// TwinCAT 3 PLC project XtsTransport
// Title: XTS Transport
// Author: D.Hauer
// ProjectVersion: 0.0.1
// Description: basic functionblocks for building XTS transport
// ProgramVersion: 3.1.4026.16
// libraries:
//   Tc2_Math, * (Beckhoff Automation GmbH)
//   Tc2_MC2, * (Beckhoff Automation GmbH)
//   Tc2_Standard, * (Beckhoff Automation GmbH)
//   Tc2_System, * (Beckhoff Automation GmbH)
//   Tc2_Utilities, * (Beckhoff Automation GmbH)
//   Tc2_XmlDataSrv, * (Beckhoff Automation GmbH)
//   Tc3_McCollisionAvoidance, * (Beckhoff Automation GmbH)
//   Tc3_McCoordinatedMotion, * (Beckhoff Automation GmbH)
//   Tc3_Module, * (Beckhoff Automation GmbH)
//   Tc3_XTS_Utility, * (Beckhoff Automation GmbH)
//   VisuDialogs, * (System)
// project tree:
//   APPLICATION/ MAIN_APP.TcPOU, fb_Simulation.TcPOU, GVL_APPLICATION.TcGVL
//   APPLICATION/_types/ E_PROCESS_CHECK.TcDUT (not stored), E_PROCESS_CTRL.TcDUT, E_PROCESS_STATE.TcDUT (not stored), ST_PROCESS_CTRL.TcDUT, ST_PROCESS_STATE.TcDUT (not stored), T_PROCESS.TcDUT
//   APPLICATION/_types/fb_Instance/ E_INSTANCE_CHECK.TcDUT (not stored), E_INSTANCE_STATE.TcDUT, fb_Instance.TcPOU
//   APPLICATION/_types/LinkedList/ fb_Process_LinkedListCtrl.TcPOU, I_Process_LinkedList.TcIO (not stored), ST_PROCESS_DATA.TcDUT (not stored), ST_PROCESS_LIST_RESULT.TcDUT
//   / GlobalTextList.TcGTLO (not stored), MAIN.TcPOU, PlcTask.TcTTO
//   MSG/ fb_LocalTime.TcPOU (not stored), f_MessageSet.TcPOU (not stored), GVL_MSG.TcGVL, MessageData.TcPOU, T_MESSAGE_LIST.TcVIS
//   MSG/types/ e_Device.TcDUT, E_MessageType.TcDUT (not stored), E_MESSAGE_STATE.TcDUT (not stored), e_Subdevice.TcDUT, ST_Message.TcDUT (not stored), TL_E_MESSAGETYPE.TcTLO (not stored)
//   XML/Configuration/ fb_Configuration.TcPOU
//   XML/Configuration/types/ E_CONFIG_CTRL.TcDUT (not stored), E_CONFIG_STATE.TcDUT (not stored), fb_XmlRead.TcPOU (not stored), fb_XmlWrite.TcPOU (not stored), ST_Configuration.TcDUT (not stored)
//   XTS/CaGroup/ FB_CaGroup.TcPOU, I_XtsTransport_CaGroup.TcIO (not stored)
//   XTS/CaGroup/types/ E_CA_GROUP_STATE.TcDUT (not stored), E_GROUP_CHECK.TcDUT (not stored), ST_GROUP_INFO.TcDUT (not stored)
//   XTS/ GVL_XTS.TcGVL, XTS_Parameter.TcGVL
//   XTS/Mover/ fb_Mover.TcPOU, fb_MoverCtrl.TcPOU (not stored), I_XtsTransport_Mover.TcIO
//   XTS/Mover/types/ E_MOVER_CTRL.TcDUT (not stored), E_MOVER_STATE.TcDUT (not stored), ST_GEAR_DATA.TcDUT (not stored), ST_MOVER_CTRL.TcDUT (not stored), ST_MOVER_INFO.TcDUT (not stored), ST_MOVER_STATE.TcDUT (not stored), ST_MOVE_DATA.TcDUT (not stored)
//   XTS/XtsStation/ fb_Station.TcPOU, I_XtsTransport_Station.TcIO (not stored)
//   XTS/XtsStation/_types/ E_STATION_CTRL.TcDUT (not stored), E_STATION_STATE.TcDUT (not stored), fb_Station_LinkedListCtrl.TcPOU (not stored), I_Station_LinkedList.TcIO (not stored), ST_STATION_CTRL.TcDUT (not stored), ST_STATION_LIST_RESULT.TcDUT (not stored), ST_STATION_MOVER_DATA.TcDUT (not stored), ST_STATION_PARAMETER.TcDUT (not stored), ST_STATION_STATE.TcDUT (not stored), T_NEST_OFFSET.TcDUT (not stored)
//   XTS/_Visualization/ GROUP_VISU.TcVIS, MOVER_VISU.TcVIS, STATION_VISU.TcVIS, Visualization Manager.TcVMO (not stored), XTS_TRANSPORT.TcVIS, XPU_VISU.TcVIS
//   XTS/_Visualization/textlists/ TL_E_CTRL_MOVER.TcTLO (not stored), TL_E_CTRL_STATION.TcTLO (not stored), TL_E_CTRL_TRANSPORT.TcTLO (not stored), TL_E_CTRL_XPU.TcTLO (not stored)
//   XTS/Xpu/ fb_Xpu.TcPOU (not stored), fb_XpuCtrl.TcPOU (not stored)
//   XTS/Xpu/types/ E_XPU_CHECK.TcDUT (not stored), E_XPU_CTRL.TcDUT (not stored), E_XPU_INIT.TcDUT (not stored), E_XPU_STATE.TcDUT (not stored), ST_XPU_CTRL.TcDUT (not stored), ST_XPU_INFO.TcDUT (not stored), ST_XPU_STATE.TcDUT (not stored)
//   XTS/XtsTransportUnit/ fb_TransportUnit.TcPOU
//   XTS/XtsTransportUnit/types/ E_XTS_TRANSPORT_CHECK.TcDUT (not stored), E_XTS_TRANSPORT_CTRL.TcDUT (not stored), E_XTS_TRANSPORT_STATE.TcDUT, ST_XTS_TRANSPORT_CTRL.TcDUT (not stored), ST_XTS_TRANSPORT_STATE.TcDUT (not stored)
//   XTS/_types/ E_PROGRESS.TcDUT, f_GetProgress.TcPOU (not stored), f_GetState.TcPOU (not stored)

CONFIGURATION XtsTransport
    RESOURCE PLC ON TwinCAT3
        TASK PlcTask(INTERVAL := T#1ms, PRIORITY := 15);
        PROGRAM MAIN WITH PlcTask : MAIN;
        PROGRAM MAIN_APP WITH PlcTask : MAIN_APP;
    END_RESOURCE
END_CONFIGURATION

// ---- APPLICATION/_types/E_PROCESS_CTRL.TcDUT
{attribute 'qualified_only'}
{attribute 'strict'}
{attribute 'to_string'}
TYPE E_PROCESS_CTRL :
(
  PROCESS_INIT              := 10,
  PROCESS_DISABLE           := 20,
  PROCESS_ENABLE            := 30,

  PROCESS_STATIONS_ENTER    := 40,
  PROCESS_STATIONS_SEND,

  PROCESS_START             := 60,
  PROCESS_DONE              := 70,
  PROCESS_STATIONS_OUTFEED  := 80
);
END_TYPE

// ---- APPLICATION/_types/fb_Instance/E_INSTANCE_STATE.TcDUT
{attribute 'qualified_only'}
{attribute 'strict'}
{attribute 'to_string'}
TYPE E_INSTANCE_STATE :
(
	INVALID,
  INIT,
  DISABLED,
  DETECT_IN_LIST,
  ENABLED,
  WORKING,
  FINISH
);
END_TYPE

// ---- APPLICATION/_types/LinkedList/ST_PROCESS_LIST_RESULT.TcDUT
TYPE ST_PROCESS_LIST_RESULT :
STRUCT
  wState    : WORD;   // wState == 0 --> all ok
  nIndex    : ULINT;
  stData    : ST_PROCESS_DATA;  // copy of list entry
END_STRUCT
END_TYPE

// ---- APPLICATION/_types/ST_PROCESS_CTRL.TcDUT
TYPE ST_PROCESS_CTRL :
STRUCT
  Cmd               : E_PROCESS_CTRL;
  ProcessTarget     : UINT;
  ActivateStation   : WORD; // every bit is a XtsStation
  NestMask          : WORD; // every bit is a PosStop in a XtsStation, one mask for all XtsStations
END_STRUCT
END_TYPE

// ---- APPLICATION/_types/T_PROCESS.TcDUT
TYPE T_PROCESS : WORD; END_TYPE

// ---- MSG/types/e_Device.TcDUT
{attribute 'to_string'}
TYPE e_Device :
(
  Device_Null,
  General           :=  1000,
  CaGroup           :=  2000,
  Xpu               :=  3000,
  XpuCtrl           :=  4000,
  Mover             :=  5000,
  MoverCtrl         :=  6000,
  XtsTransportUnit  :=  7000,
  XfcTriggerBox     :=  8000,
  XfcTouchProbe     :=  9000,
  XtsStation        := 10000,

  Camming           := 11000,
  NciChannel        := 12000,
  NciChannelCtrl    := 13000,
  Axis              := 14000,
  XfcAxis           := 15000,
  Data              := 16000,

  Process           := 20000,
  Application       := 30000
)UDINT;
END_TYPE

// ---- MSG/types/e_Subdevice.TcDUT
{attribute 'strict'}
{attribute 'to_string'}
TYPE e_Subdevice :
(
  // sub device for message system
  General                 :=  0,
  // Motion Control FB Instances
  fbPower,
  fbReset,
  fbResetSercos,
  fbHalt,
  fbStop,                 // 5
  fbHome,
  fbJog,
  fbMoveVelocity1,
  fbMoveVelocity2,
  fbMoveAbsolute1,        // 10
  fbMoveAbsolute2,
  fbMoveEndless,
  fbMovePtP,

  // CA CollisionAvoidance FB instances
  // CA group fb instances
  fbCaGroup             := 30,
  fbMoveToPosCa,
  fbSendToAbsPosCa,
  fbSendToModuloPosCa,
  fbGearInPosCa,
  fbGroupAddAxis,
  fbGroupRemoveAxis,
  fbGroupDisable,
  fbGroupEnable,
  fbGroupErrorRead,
  fbGroupStatusRead,
  fbGroupReset,
  fbGroupStop,

  fbGearIn                := 50,
  fbGearOut,
  fbGearInMultiMaster,

  fbCamIn                 := 60,
  fbCamOut,

  fbCamOutV2              := 80,
  fbCamInV2,
  fbCamScalingV2,
  fbCamInfoV2,
  fbReadMotionFunction,
  fbReadMotionFunctionPoint,
  fbReadMotionFunctionValues,
  fbWriteMotionFunction,
  fbWriteMotionFunctionPoint,
  fbSetOnlineChangeMode,

  fbReadParameter         := 100,
  fbReadBoolParameter,
  fbWriteParameter,
  fbWriteBoolParameter,

  fbBuildGroup            := 200,
  fbClearGroup,
  fbLoadProg,
  fbResetItp,
  fbStartStopItp,
  fbEStopItp,             // 205
  fbStepOnAfterEStopItp,
  fbConfirmHskItp,
  fbDelDtgItp,
  fbNciFeedTablePreparation,
  fbNciFeedTable,         // 210
  fbReadLine,
  fbItpReadRParams,
  fbItpWriteRParams,
  Get_ItpState,
  Get_Error,              // 215


  XfcPositionAtTime       := 300,
  XfcTimeOfPosition,
  XfcTimeToPosition,
  XfcTimeToModuloPosition,
  XfcRecordedPosition,
  XfcTouchProbe,          // 305
  XfcTouchProbeEL1258,
  XfcTouchProbeOptions,
  XfcTriggerRef,
  XfcTriggerRef_MT,
  XfcEl1258Interface_MT,  // 310
  XfcRecordedPosition_MT,
  XfcTriggerOut,
  XfcTriggerStart,
  XfcSwitchOn_2252,
  XfcSwitchOff_2252,      // 315
  XfcInit,
  XfcLatchPosition,
  XfcWaitForPosition,

  AxisMode              := 1000,
  AxisControl,

  NciControl            := 2000,
  NciStartUp,
  NciCycle,
  NciIdle,

  StationLinkedList     := 3000,
  StationInitList,
  StationAddHead,
  StationAddTail,
  StationGetHead,
  StationRemoveHeadValue,

  StationControl        := 4000,
  StationState, 

  Xpu_fbEnvironment     := 5000,
  Xpu_fbProcessingUnit,
  Xpu_fbXpuPart,
  Xpu_fbXpuTrack,
  Xpu_fbMc2CaGroup,

  Xpu_fbPartModules     := 5500,

  Xpu_fbMoverXpu        := 6000,

  CamControl            := 8000,
  CamStartUp,
  CamCycle,

  Process_StationCollector    := 11000,
  Process_Process_Collector   := 11100,
  Process_ProcessCollector_Init,
  Process_ProcessCollector_Cycle,
  Process_ProcessCollector_Control,

  Process_LinkedList_GetHead,
  Process_LinkedList_RemoveHead,
  Process_LinkedList_AddTail,

  Process_BufferInfeed
)DINT;
END_TYPE

// ---- XTS/XtsTransportUnit/types/E_XTS_TRANSPORT_STATE.TcDUT
{attribute 'to_string'}
TYPE E_XTS_TRANSPORT_STATE :
(
  TRANSPORT_NULL,
  TRANSPORT_INVALID,
  TRANSPORT_INIT            := 10,  // Xpu, Group, Mover initialization: init TcCOM objects, clear errors, clear group, check Xpu data, check mover detection
  TRANSPORT_IDLE,                   // cyclic check for errors, check Xpu data

  TRANSPORT_MOVER_ENABLE    := 20,  // all mover are enabled, checked for ControlLoopClosed
  TRANSPORT_MOVER_DISABLE,          // all mover are disabled
  TRANSPORT_MOVER_HALT_CA,          // all mover standstill

  TRANSPORT_GROUP_CLEAR     := 30,  // halt all movers, clear errors, remove all movers from group, clear group
  TRANSPORT_GROUP_BUILD,            // add all movers to group
  TRANSPORT_GROUP_ENABLE,           // group with movers is enabled
  TRANSPORT_GROUP_STOP,             // CaGroup Stop, CaGroup Reset, All movers halt

  TRANSPORT_START           := 40,  // move all mover[i] to start position
  TRANSPORT_RESTART                 // move all mover[i] to LastPosition[i]
)UINT;
END_TYPE

// ---- XTS/_types/E_PROGRESS.TcDUT
{attribute 'qualified_only'}
//{attribute 'strict'}
{attribute 'to_string'}
TYPE E_PROGRESS :
(
  // progress is used in project to mirror state of requested command/function
  PROGRESS_INVALID,
  PROGRESS_NOT_EXIST      :=   100,
  PROGRESS_INIT           :=  1000,
  PROGRESS_BUSY           :=  2000,
  PROGRESS_PREPARE        :=  3000,
  PROGRESS_STARTUP        :=  4000,
  PROGRESS_CHECK          :=  5000,
  PROGRESS_OCCUPIED       :=  6000,
  PROGRESS_WORKING        :=  7000,
  PROGRESS_STILL_WORKING  :=  8000,
  PROGRESS_ERROR          :=  9000,
  PROGRESS_DONE           := 10000
)UINT;
END_TYPE

// ---- APPLICATION/GVL_APPLICATION.TcGVL
VAR_GLOBAL CONSTANT
  MAX_PROCESS       : UINT := 11;
END_VAR
{attribute 'qualified_only'}
VAR_GLOBAL
  Simulation        : ARRAY[1..MAX_PROCESS] OF fb_Simulation;
END_VAR

// ---- MSG/GVL_MSG.TcGVL
{attribute 'qualified_only'}
VAR_GLOBAL CONSTANT
  //-----------------------------------------------------------------------------
  // file paths for message system
  //  - compiler define option WIN switches to Windows file paths
  //-----------------------------------------------------------------------------
{IF defined (WIN)}
  {info 'WIN folders'}
  LOG_DIR               : STRING  := 'C:\TwinCAT\#MsgFiles\';
  CONFIG_DIR            : STRING  := 'C:\TwinCAT\XPU_PLC_StationConfig\';
{ELSE}
  {info 'BSD folders'}
  LOG_DIR               : STRING  := '/usr/local/etc/TwinCAT/#MsgFiles/';
  CONFIG_DIR            : STRING  := '/usr/local/etc/TwinCAT/XPU_PLC_StationConfig/';
{END_IF}

  LOG_FILE              : STRING  := 'MSG_XtsTransport_';
  CONFIG_FILE           : STRING  := 'Config_XPU_'; // OTCID of fb_Environment is added to name on writing

  MAX_MESSAGE           : UINT    := 200; // max entry in message list
END_VAR
VAR_GLOBAL
  Messages                        : ARRAY[1..MAX_MESSAGE] OF ST_Message;
  MessageIndex                    : UINT := 1; // message index
  MessageError                    : UINT := 0; // error counter

  fbLocalTime                     : fb_LocalTime;
  dtLocalTime                     : DT;
  sLocalTime                      : STRING;

  MessageLevelXpu                 : E_MessageType;
  MessageLevelStations            : ARRAY[1..MAX_STATION] OF E_MessageType;
  MessageLevelMovers              : ARRAY[1..MAX_MOVER]   OF E_MessageType;

  MessageLevelProcess             : ARRAY[1..MAX_PROCESS] OF E_MessageType;

{IF defined (TEST)}
  {info 'TEST logging enabled'}
  MessageLevel                    : E_MessageType := eMessageVerbose; // a lot of messages
{ELSE}
  MessageLevel                    : E_MessageType := eMessageError;    // not as much messages 
{END_IF}

END_VAR

// ---- XTS/GVL_XTS.TcGVL
{attribute 'qualified_only'}
VAR_GLOBAL
  //---------------------------------------------------------------------------
  // XTS Station
  //  - handshakes mover in station with extern control
  //  - station parameters (positions, gap, dyn. constraints, description...)
  StationStart        : ST_STATION_PARAMETER;   // Xts transport is sending all mover to this position (CMD_TRANSPORT_START)
  StationStartIndex   : UINT := 1;              // index of XtsStation where all movers are entered into linked list.

  // station handshaking with mover and extern process
  // station sends mover to target station/WaitPos
  // station adds mover data to LinkedList.AddTail() of target station
  Station             : ARRAY[1..MAX_STATION] OF fb_Station;
  StationList         : ARRAY[1..MAX_STATION] OF fb_Station_LinkedListCtrl;

  StationQueue        : ARRAY[1..MAX_STATION]    OF 
                        ARRAY[1..MAX_LIST_NODES] OF ST_STATION_MOVER_DATA;

  // interface for access to List methods
  StationListItf      : ARRAY[1..MAX_STATION] OF I_Station_LinkedList;

  // interface for access to station methods
  StationCtrlItf      : ARRAY[1..MAX_STATION] OF I_XtsTransport_Station;

  // ctrl / state datafields for extern control
  StationCtrl         : ARRAY[1..MAX_STATION] OF ST_STATION_CTRL;   // control for extern to write
  StationState        : ARRAY[1..MAX_STATION] OF ST_STATION_STATE;  // state for extern to read

  // station parameter
  StationParameter    : ARRAY[1..MAX_STATION] OF ST_STATION_PARAMETER; // XtsStation (fb_Station) positions and dyn constraints

  // static position offsets in stations
  PositionOffset      : ARRAY[1..MAX_STATION] OF T_NEST_OFFSET; // added to PosStop[] in XtsStation


  //---------------------------------------------------------------------------
  // XTS
  // XTS TransportUnit
  //  - handles request for XPU, Group, Mover, StartUp, ReStart
  XtsTransport        : fb_TransportUnit;         // manages members of XTS transport for extern to access

  XtsTransportCtrl    : ST_XTS_TRANSPORT_CTRL;    // control of XTS transport for extern to write
  XtsTransportState   : ST_XTS_TRANSPORT_STATE;   // state   of XTS transport for extern to read


  //---------------------------------------------------------------------------
  // XPU
  // XTS-Utility checks
  // XTS-Utility interfaces for you to use
  Xpu             : fb_XpuCtrl;

  XpuCtrl         : ST_XPU_CTRL;
  XpuState        : ST_XPU_STATE;
  XpuInfo         : ST_XPU_INFO;
  XpuModules      : ARRAY[1..MAX_MODULE] OF Tc3_XTS_Utility.ST_InfoDataView;


  //---------------------------------------------------------------------------
  // Collision avoidance group CA
  //
  // - add mover to group
  // - build group
  // - clear group
  CaGroup         : FB_CaGroup;                   // cyclic check of CaGroup state and errors; carries methods for handling CaGroup
  CaGroupItf      : I_XtsTransport_CaGroup;       // Interface used by fb_TransportUnit

  // cyclic mapping to MOTION/Objects/CaGroup 
  CaGroupRef      : Tc3_McCoordinatedMotion.AXES_GROUP_REF;

  // Info data from CaGroup FB
  CaGroupInfo     : ST_GROUP_INFO;                // cyclic info about CaGroup for fb_TransportUnit to read
  //---------------------------------------------------------------------------

  //---------------------------------------------------------------------------
  // MC2 encapsulation, CA movement
  Mover           : ARRAY[1..MAX_MOVER] OF fb_MoverCtrl;    // MC and CA methods for mover; cyclic check for individual command on mover

  MoverCtrl       : ARRAY[1..MAX_MOVER] OF ST_MOVER_CTRL;   // control of individual mover for extern to write
  MoverState      : ARRAY[1..MAX_MOVER] OF ST_MOVER_STATE;  // state   of individual mover for extern to read

  MoverItf        : ARRAY[1..MAX_MOVER] OF I_XtsTransport_Mover;  // Interface used by fb_TransportUnit

  LastPosition    : ARRAY[1..MAX_MOVER] OF LREAL;           // on execute of any movement, value is saved here (used by fb_Mover)
  LastGap         : ARRAY[1..MAX_MOVER] OF LREAL;           // on execute of any movement, value is saved here (used by fb_Mover)

  MoverInfo       : ARRAY[1..MAX_MOVER] OF ST_MOVER_INFO;   // cyclic info about mover for extern to read

  MoveData        : ARRAY[1..MAX_MOVER] OF ST_MOVE_DATA;    // dynamic constraints for move commands
  GearData        : ARRAY[1..MAX_MOVER] OF ST_GEAR_DATA;    // dynamic constraints and positions for GearIn/GearInPosCa
  
  // cyclic mapping to MOTION/Axes
  AxisRefMover    : ARRAY[1..MAX_MOVER] OF Tc2_MC2.AXIS_REF;
  //---------------------------------------------------------------------------

  //---------------------------------------------------------------------------
  // XML configuration helper
  XmlConfiguration   : fb_Configuration;


END_VAR

// ---- XTS/XTS_Parameter.TcGVL
//{attribute 'qualified_only'}
VAR_GLOBAL CONSTANT
// HAUD 2025 08 09
//
//    XTS_TRANSPORT_LAYER project
//    
//    MIT License
//    
//    Copyright (c) 2025 HAUD
//    
//    Permission is hereby granted, free of charge, to any person obtaining a copy
//    of this software and associated documentation files (the "Software"), to deal
//    in the Software without restriction, including without limitation the rights
//    to use, copy, modify, merge, publish, distribute, sublicense, and/or sell
//    copies of the Software, and to permit persons to whom the Software is
//    furnished to do so, subject to the following conditions:
//    
//    The above copyright notice and this permission notice shall be included in all
//    copies or substantial portions of the Software.
//    
//    THE SOFTWARE IS PROVIDED "AS IS", WITHOUT WARRANTY OF ANY KIND, EXPRESS OR
//    IMPLIED, INCLUDING BUT NOT LIMITED TO THE WARRANTIES OF MERCHANTABILITY,
//    FITNESS FOR A PARTICULAR PURPOSE AND NONINFRINGEMENT. IN NO EVENT SHALL THE
//    AUTHORS OR COPYRIGHT HOLDERS BE LIABLE FOR ANY CLAIM, DAMAGES OR OTHER
//    LIABILITY, WHETHER IN AN ACTION OF CONTRACT, TORT OR OTHERWISE, ARISING FROM,
//    OUT OF OR IN CONNECTION WITH THE SOFTWARE OR THE USE OR OTHER DEALINGS IN THE
//    SOFTWARE.

  Version             : STRING  := '4.00.11';

  MAX_MOVER           : UINT    := TO_UINT(Tc3_XTS_Utility.TcIoXtsEnvironmentParameterList.MaxXtsMoversPerXpu);
  MAX_MODULE          : UINT    := TO_UINT(Tc3_XTS_Utility.TcIoXtsEnvironmentParameterList.MaxModulesPerPart);
  MAX_PART            : UINT    := TO_UINT(Tc3_XTS_Utility.TcIoXtsEnvironmentParameterList.MaxXtsPartsPerXpu);
  MAX_TRACK           : UINT    := TO_UINT(Tc3_XTS_Utility.TcIoXtsEnvironmentParameterList.MaxXtsTracksPerXpu);
  MAX_GROUP           : UINT    := TO_UINT(Tc3_XTS_Utility.TcIoXtsEnvironmentParameterList.MaxXtsCaGroup);

  MAX_INFO_SERVER     : UINT    := TO_UINT(Tc3_XTS_Utility.TcIoXtsEnvironmentParameterList.MaxXtsInfoServer);
  MAX_INFO_STATION    : UINT    := TO_UINT(Tc3_XTS_Utility.TcIoXtsEnvironmentParameterList.MaxXtsInfoStation);
  MAX_INFO_STOP_POS   : UINT    := TO_UINT(Tc3_XTS_Utility.TcIoXtsEnvironmentParameterList.MaxXtsStopPositionsPerStation);

  MAX_PARAMETER_SET   : UINT    := TO_UINT(Tc3_XTS_Utility.TcIoXtsEnvironmentParameterList.MaxXtsParameterSet);

  MAX_NCT_BASE_UNIT   : UINT    := TO_UINT(Tc3_XTS_Utility.TcIoXtsEnvironmentParameterList.MaxXtsNctBaseUnitInterfaces);

  MAX_STATION         : UINT    := 22;

  MAX_STATION_NEST    : UINT    := TO_UINT(SIZEOF(ST_STATION_STATE.nMask)*8);
  // MAX_LIST_NODES      : UINT    := MAX_MOVER;
  MAX_LIST_NODES      : UINT    := 32; // visualization can not handle access to MAX_MOVER
  MAX_MASTER          : UINT    := 1;
END_VAR

// ---- XTS/Mover/I_XtsTransport_Mover.TcIO
INTERFACE I_XtsTransport_Mover

METHOD Disable : E_PROGRESS
VAR_INPUT
  Execute             : BOOL;
END_VAR
END_METHOD

METHOD Enable : E_PROGRESS
VAR_INPUT
  Execute             : BOOL;
END_VAR
END_METHOD

METHOD GearIn : E_PROGRESS;
VAR_INPUT
  Execute             : BOOL;
  stMoveData          : ST_MOVE_DATA;
  stGearData          : ST_GEAR_DATA;
END_VAR
END_METHOD

METHOD GearInPosCa : E_PROGRESS
VAR_INPUT
  Execute             : BOOL;
  stMoveData          : ST_MOVE_DATA;
  stGearData          : ST_GEAR_DATA;  
END_VAR
END_METHOD

METHOD GearOut : E_PROGRESS
VAR_INPUT
  Execute             : BOOL;
END_VAR
END_METHOD

METHOD Halt : E_PROGRESS
VAR_INPUT
  Execute             : BOOL;
  stMoveData          : ST_MOVE_DATA;
END_VAR
END_METHOD

METHOD HaltCa : E_PROGRESS
VAR_INPUT
  Execute             : BOOL;
  stMoveData          : ST_MOVE_DATA;
END_VAR
END_METHOD

PROPERTY MessageLevel : e_messagetype
SET
END_SET
END_PROPERTY

PROPERTY ModuloTurn : dint
GET
END_GET
END_PROPERTY

METHOD MoveToPos : E_PROGRESS
VAR_INPUT
  Execute             : BOOL;
  stMoveData          : ST_MOVE_DATA;
END_VAR
END_METHOD

METHOD MoveToPosCa : E_PROGRESS
VAR_INPUT
  Execute             : BOOL;
  stMoveData          : ST_MOVE_DATA;
END_VAR
END_METHOD

PROPERTY RailLength : LREAL
GET
END_GET
SET
END_SET
END_PROPERTY

METHOD Reset : E_PROGRESS
VAR_INPUT
  Execute             : BOOL;
END_VAR
END_METHOD

METHOD SendToAbsPosCa : E_PROGRESS
VAR_INPUT
  Execute             : BOOL;
  stMoveData          : ST_MOVE_DATA;
END_VAR
END_METHOD

METHOD SendToModuloPosCa : E_PROGRESS
VAR_INPUT
  Execute             : BOOL;
  stMoveData          : ST_MOVE_DATA;
END_VAR
END_METHOD

METHOD Stop : E_PROGRESS
VAR_INPUT
  Execute             : BOOL;
  stMoveData          : ST_MOVE_DATA;
END_VAR
END_METHOD

END_INTERFACE

// ---- MAIN.TcPOU
//---------------------------------------------------------------------------------------------------------------
//
//  HAUD 2024.03.18
//
//  - XTS_TRANSPORT_LAYER
//  - transport layer members:
//    - CaGroup
//      - access to Group functions
//
//    - Mover
//      - access to MC and CA motion functions
//
//    - Xpu (ProcessingUnit)
//      - access to TcCOM Objects in Environment
//
//    - Transport Control Unit
//      - coordinates members to get XTS in defined states
//
//    - Xts Stations
//      - handshakes with extern control for mover transport
//
//  - global datafields for mrmbers in GVL_XTS namespace
//  - global interface datafields for use in members
//  - structures are assigned by reference for every member
//
//---------------------------------------------------------------------------------------------------------------
// HAUD 2024 05 29
//
//    XTS_TRANSPORT_LAYER project
//    
//    MIT License
//    
//    Copyright (c) 2024 HAUD
//    
//    Permission is hereby granted, free of charge, to any person obtaining a copy
//    of this software and associated documentation files (the "Software"), to deal
//    in the Software without restriction, including without limitation the rights
//    to use, copy, modify, merge, publish, distribute, sublicense, and/or sell
//    copies of the Software, and to permit persons to whom the Software is
//    furnished to do so, subject to the following conditions:
//    
//    The above copyright notice and this permission notice shall be included in all
//    copies or substantial portions of the Software.
//    
//    THE SOFTWARE IS PROVIDED "AS IS", WITHOUT WARRANTY OF ANY KIND, EXPRESS OR
//    IMPLIED, INCLUDING BUT NOT LIMITED TO THE WARRANTIES OF MERCHANTABILITY,
//    FITNESS FOR A PARTICULAR PURPOSE AND NONINFRINGEMENT. IN NO EVENT SHALL THE
//    AUTHORS OR COPYRIGHT HOLDERS BE LIABLE FOR ANY CLAIM, DAMAGES OR OTHER
//    LIABILITY, WHETHER IN AN ACTION OF CONTRACT, TORT OR OTHERWISE, ARISING FROM,
//    OUT OF OR IN CONNECTION WITH THE SOFTWARE OR THE USE OR OTHER DEALINGS IN THE
//    SOFTWARE.
//---------------------------------------------------------------------------------------------------------------
PROGRAM MAIN
VAR
	bInit 				: BOOL;
  eInit         : E_PROGRESS;

  nStation,
	nMover,
  nMoverSelected,
  nStationSelected,
  nStationParameter   : UINT;

  sStationText        : STRING(30);

  eTransportState     : E_XTS_TRANSPORT_STATE;
  eTransportResult    : E_PROGRESS;

  eXpuState           : E_XPU_STATE;
  eXpuResult          : E_PROGRESS;
  eXpuCheck           : E_XPU_CHECK;

  eMoverState         : E_MOVER_STATE;
  eMoverResult        : E_PROGRESS;

  sCaGroupState,
  sTransportState,
  sTransportCheck,
  sTransportResult,
  sXpuState,
  sXpuResult,
  sXpuCheck,
  sXpuOpMode,
  sXpuMoverdetectionMode,
  sXpuMoverAssignement,
  sMoverState,
  sMoverResult,
  sStationState,
  sStationStateMask,
  sStationCtrlMask        : STRING;

  bStationEnable,
  bStationEnter,
  bStationStart,
  bStationDone,
  bStationOut,
  bStationGone            : BOOL;

  tStationSelectedQueue   : ARRAY[1..MAX_LIST_NODES] OF ST_STATION_MOVER_DATA;

  tonWriteLog             : Tc2_Standard.TON;
  tWriteLog               : TIME := T#5S;

  nStn                    : UINT;
END_VAR

//############################################################################
// Local time; used for timestamps
//############################################################################
GVL_MSG.fbLocalTime(
                    sLocalTime          => GVL_MSG.sLocalTime, 
                    dtLocalTime         => GVL_MSG.dtLocalTime);
//############################################################################

//############################################################################
// 	example for init sequence
//############################################################################	
IF NOT bInit
THEN
  CASE eInit
  OF
    E_PROGRESS.PROGRESS_INVALID,
    E_PROGRESS.PROGRESS_DONE:         // clear command interface
      eInit                                   := E_PROGRESS.PROGRESS_BUSY;
      GVL_XTS.XpuCtrl.Cmd                     := E_XPU_CTRL.XTS_CMD_NULL;
      GVL_MSG.MessageLevelXpu                 := GVL_MSG.MessageLevel;
      GVL_XTS.CaGroup.MessageLevel            := GVL_MSG.MessageLevel;
      FOR nStation := 1 TO MAX_STATION
      DO
        GVL_MSG.MessageLevelStations[nStation]:= GVL_MSG.MessageLevel;
      END_FOR
      FOR nMover := 1 TO MAX_MOVER
      DO
        GVL_MSG.MessageLevelMovers[nMover]    := GVL_MSG.MessageLevel;
      END_FOR


    E_PROGRESS.PROGRESS_BUSY:         // init Xpu, ProcessingUnit, MotorModules
      eInit                                   := E_PROGRESS.PROGRESS_PREPARE;
      GVL_XTS.XpuCtrl.Cmd                     := E_XPU_CTRL.XTS_CMD_INIT;

    E_PROGRESS.PROGRESS_PREPARE:      // wait for init to be done
      IF (GVL_XTS.XpuState.State      = E_XPU_STATE.XTS_INIT + E_PROGRESS.PROGRESS_DONE)
      THEN
        eInit                                 := E_PROGRESS.PROGRESS_STARTUP;
        GVL_XTS.XpuCtrl.Cmd                   := E_XPU_CTRL.XTS_IDLE;
      END_IF

    E_PROGRESS.PROGRESS_STARTUP:      // assign mover interfaces
      eInit                                   := E_PROGRESS.PROGRESS_CHECK;
      FOR nMover := 1 TO MAX_MOVER
      DO
        GVL_XTS.MoverItf[nMover]              := GVL_XTS.Mover[nMover];
      END_FOR

    E_PROGRESS.PROGRESS_CHECK:        // assign CaGroup interface
      eInit                                   := E_PROGRESS.PROGRESS_OCCUPIED;
      GVL_XTS.CaGroupItf                      := GVL_XTS.CaGroup;

    E_PROGRESS.PROGRESS_OCCUPIED:     // StartStation for XtsTransportCtrl.Cmd := E_XTS_TRANSPORT_CTRL.CMD_TRANSPORT_START;
      eInit                                   := E_PROGRESS.PROGRESS_WORKING;
      // where to start?
      GVL_XTS.XtsTransport.StationStartIndex  := 1;

      StationParameterInit();


    E_PROGRESS.PROGRESS_WORKING:
      // Start Position parameters
      GVL_XTS.StationStart.rPosWait           :=    GVL_XTS.StationParameter[GVL_XTS.XtsTransport.StationStartIndex].rPosWait -10.0; // this value may differ from the GVL_XTS.StationParameter[StartStationIndex], IF it differs, you MUST have room for positive movement to GVL_XTS.StationParameter[StartStationIndex].rWaitPos
      GVL_XTS.StationStart.rGap               :=    105.0; // may differ, or just copy from GVL_XTS.StationParameter[StartStationIndex]
      GVL_XTS.StationStart.rVelo              :=    750.0; // may differ, or just copy from GVL_XTS.StationParameter[StartStationIndex]
      GVL_XTS.StationStart.rAccDec            :=  12000.0; // may differ, or just copy from GVL_XTS.StationParameter[StartStationIndex]
      GVL_XTS.StationStart.rJerk              := 400000.0; // may differ, or just copy from GVL_XTS.StationParameter[StartStationIndex], the movements are more robust if you keep this value in a narrow range, since jumps lead to adjusting movements within the CA Group

      IF (GVL_XTS.XtsTransport.StationStartIndex > 0) AND
         (GVL_XTS.XtsTransport.StationStartIndex < MAX_STATION+1)
      THEN
        GVL_XTS.StationStart.nConfiguredStopCount := GVL_XTS.StationParameter[GVL_XTS.XtsTransport.StationStartIndex].nConfiguredStopCount;
      END_IF

      bInit                                           := TRUE;
      eInit                                           := E_PROGRESS.PROGRESS_DONE;
  END_CASE
END_IF

//############################################################################
// 	XTS Transport Unit
//############################################################################
//  - main control function block for transport layer
//  - requires access to member controls
//    - Xpu
//    - CaGroup
//    - Mover
//    - Station Control
//    - Station LinkedList Interface
//############################################################################
//
// cyclic call
GVL_XTS.XtsTransport();

// main control
GVL_XTS.XtsTransport.Ctrl               REF= GVL_XTS.XtsTransportCtrl;   // main control
GVL_XTS.XtsTransport.State              REF= GVL_XTS.XtsTransportState;  // main state
                                        
// member controls                      
GVL_XTS.XtsTransport.XpuCtrl            REF= GVL_XTS.XpuCtrl;
GVL_XTS.XtsTransport.XpuState           REF= GVL_XTS.XpuState;
GVL_XTS.XtsTransport.XpuInfo            REF= GVL_XTS.XpuInfo;
                                        
GVL_XTS.XtsTransport.GroupItf           :=   GVL_XTS.CaGroupItf;
GVL_XTS.XtsTransport.GroupInfo          REF= GVL_XTS.CaGroupInfo;
                                        
GVL_XTS.XtsTransport.MoverItf           REF= GVL_XTS.MoverItf;
GVL_XTS.XtsTransport.MoverInfo          REF= GVL_XTS.MoverInfo;
GVL_XTS.XtsTransport.MoverLastPosition  REF= GVL_XTS.LastPosition;
GVL_XTS.XtsTransport.MoverLastGap       REF= GVL_XTS.LastGap;
                                        
GVL_XTS.XtsTransport.StationStart       REF= GVL_XTS.StationStart;      // start position for E_XTS_TRANSPORT_CTRL.CMD_TRANSPORT_START
GVL_XTS.XtsTransport.StationCtrlItf     REF= GVL_XTS.StationCtrlItf;    // station interfaces are required for accessing station methods
GVL_XTS.XtsTransport.StationListsItf    REF= GVL_XTS.StationListItf;    // list interface is required for access to linked list methods
GVL_XTS.XtsTransport.StationControl     REF= GVL_XTS.StationCtrl;
GVL_XTS.XtsTransport.StationState       REF= GVL_XTS.StationState;
//############################################################################



//############################################################################
// 	XTS Stations
//############################################################################	
FOR nStation := 1 TO MAX_STATION
DO
  GVL_XTS.Station[nStation].StationId   := nStation;
  GVL_XTS.Station[nStation].MessageLevel:= GVL_MSG.MessageLevelStations[nStation];

  GVL_XTS.StationListItf[nStation]      := GVL_XTS.StationList[nStation];   // interfaces for list methods
  GVL_XTS.StationCtrlItf[nStation]      := GVL_XTS.Station[nStation];       // interfaces for station methods

  GVL_XTS.Station[nStation].Ctrl        REF= GVL_XTS.StationCtrl;           // station ctrl from extern
  GVL_XTS.Station[nStation].State       REF= GVL_XTS.StationState;          // station state to extern

  GVL_XTS.Station[nStation].ItfStations REF= GVL_XTS.StationListItf;        // give every station all list interfaces for writing mover tickets
  GVL_XTS.Station[nStation].ItfMover    REF= GVL_XTS.MoverItf;              // give every station all mover interfaces for movement in / out of station
  GVL_XTS.Station[nStation].Mover       REF= GVL_XTS.AxisRefMover;          // AXIS_REF to read infos from
  GVL_XTS.Station[nStation].MoverOffset REF= GVL_XTS.PositionOffset;        // static offsets for all stations, all movers, all stop positions


  GVL_XTS.Station[nStation].StationParameter  REF= GVL_XTS.StationParameter;// give every station all station parameters for sending to WaitPos of target station

  // cyclic call
  GVL_XTS.Station[nStation].Cycle();                                        // cycle for handshaking with extern

  // Queue data for each station
  GVL_XTS.StationQueue[nStation]        := GVL_XTS.StationListItf[nStation].Data;
END_FOR
//############################################################################



//############################################################################
// 	XPU environment
//############################################################################	
GVL_XTS.Xpu.XpuInstance               :=   1;
GVL_XTS.Xpu.MessageLevel              :=   GVL_MSG.MessageLevelXpu;

GVL_XTS.Xpu.Ctrl                      REF= GVL_XTS.XpuCtrl;
GVL_XTS.Xpu.State                     REF= GVL_XTS.XpuState;
GVL_XTS.Xpu.XpuModuleInfoData         REF= GVL_XTS.XpuModules;

GVL_XTS.Xpu.CaGroupOID                :=   GVL_XTS.CaGroup.GroupInfo.CaGroupOID;

// cyclic call
GVL_XTS.Xpu();
GVL_XTS.XpuInfo                       :=   GVL_XTS.Xpu.XpuInfo;
//############################################################################


//############################################################################	
// 	CA-Group Class
//############################################################################	
// assignment
GVL_XTS.CaGroup.AxisRef               REF= GVL_XTS.AxisRefMover;
// Interface to Mover methods
GVL_XTS.CaGroup.MoverItf              REF= GVL_XTS.MoverItf; 

GVL_XTS.CaGroup.GroupRef              REF= GVL_XTS.CaGroupRef;

// cyclic call
GVL_XTS.CaGroup.InfoCycle(TRUE); // read group status

// InfoData from group
GVL_XTS.CaGroupInfo                   :=   GVL_XTS.CaGroup.GroupInfo;

// Interface of CaGroup
GVL_XTS.CaGroupItf                    :=   GVL_XTS.CaGroup;
//############################################################################


//############################################################################
// Mover Class	
//############################################################################	
FOR nMover := 1 TO MAX_MOVER
DO
  GVL_XTS.Mover[nMover].MoverId       :=   nMover;
  GVL_XTS.Mover[nMover].RailLength    :=   GVL_XTS.Xpu.RailLength;  // mover needs RailLength, in order to calc absolute position from modulo input
  GVL_XTS.Mover[nMover].MessageLevel  :=   GVL_MSG.MessageLevelMovers[nMover];

  GVL_XTS.Mover[nMover].Ctrl          REF= GVL_XTS.MoverCtrl;       // mover control from extern
  GVL_XTS.Mover[nMover].State         REF= GVL_XTS.MoverState;      // mover state to extern

  GVL_XTS.Mover[nMover].MoveData      REF= GVL_XTS.MoveData;        // dyn constraints for extern to write
  GVL_XTS.Mover[nMover].GearData      REF= GVL_XTS.GearData;        // GearIn/GearInPosCa data fro extern to write

  // assignment	
  GVL_XTS.Mover[nMover].Mover         REF= GVL_XTS.AxisRefMover[nMover];  // axis reference to Mover function block
  GVL_XTS.Mover[nMover].LastGap       REF= GVL_XTS.LastGap[nMover];       // reference to last used gap value datafield
  GVL_XTS.Mover[nMover].LastPosition  REF= GVL_XTS.LastPosition[nMover];  // reference to last position datafield

  GVL_XTS.Mover[nMover].MoverInfo		  REF= GVL_XTS.MoverInfo[nMover];     // refernence to mover info data (ActPos, SetPos, ...)

  GVL_XTS.MoverItf[nMover]            :=   GVL_XTS.Mover[nMover];

  // cyclic call
  GVL_XTS.Mover[nMover].Cycle();  // call AXIS_REF()
  GVL_XTS.Mover[nMover]();        // call Ctrl/State
END_FOR


//############################################################################


//############################################################################
// /logging
//############################################################################
tonWriteLog(IN:= TRUE, PT := tWriteLog);

IF (tonWriteLog.Q)
THEN
  MessageData.bWriteFile      := TRUE;
  tonWriteLog(IN:= FALSE);
END_IF

//-----------------------------------------------------------------------------------------------------------------
// write message list to file
//-----------------------------------------------------------------------------------------------------------------
MessageData(pList			        := ADR(GVL_MSG.Messages),
			      pLocalTime        := ADR(GVL_MSG.dtLocalTime), 
			      bBusy=> );

// clear write trigger
IF MessageData.bWriteFile AND
   MessageData.bDone
THEN
  MessageData.bWriteFile      := FALSE;
END_IF
//############################################################################
// logging/
//############################################################################



//############################################################################
// \xml config 
//    no startup read 
//    for manual use only
//############################################################################
GVL_XTS.XmlConfiguration.StationData   := ADR(GVL_XTS.StationParameter);
GVL_XTS.XmlConfiguration.Identity      := GVL_XTS.Xpu.XpuOtcid;
GVL_XTS.XmlConfiguration();
//############################################################################
// xml config/
//############################################################################


//############################################################################
// Visualization data	
//############################################################################	
// get enumerations from XPU for visu:
eTransportState                       := f_GetState   (GVL_XTS.XtsTransportState.State);
eTransportResult                      := f_GetProgress(GVL_XTS.XtsTransportState.State);

eXpuState                             := f_GetState   (GVL_XTS.XpuState.State);
eXpuResult                            := f_GetProgress(GVL_XTS.XpuState.State);

eXpuCheck                             := GVL_XTS.XpuState.Check;

// display xpu state and result in visu
// get strings and info
sCaGroupState                         := TO_STRING(GVL_XTS.CaGroupInfo.CaGroupState);

sTransportState                       := TO_STRING(eTransportState);
sTransportCheck                       := TO_STRING(GVL_XTS.XtsTransportState.Check);
sTransportResult                      := TO_STRING(eTransportResult);

sXpuState                             := TO_STRING(eXpuState);
sXpuResult                            := TO_STRING(eXpuResult);
sXpuCheck                             := TO_STRING(eXpuCheck);

sXpuOpMode                            := GVL_XTS.Xpu.OpModeToString();
sXpuMoverdetectionMode                := GVL_XTS.Xpu.IdDetectionModeToString();
sXpuMoverAssignement                  := GVL_XTS.Xpu.MoverPositionAssignementToString();

nMoverSelected                        := SEL((nMoverSelected<1), nMoverSelected, 1);
nMoverSelected                        := SEL((nMoverSelected>MAX_MOVER), nMoverSelected, MAX_MOVER);

nStationSelected                      := SEL((nStationSelected<1), nStationSelected, 1);
nStationSelected                      := SEL((nStationSelected>MAX_STATION), nStationSelected, MAX_STATION);

bStationEnable                        := SEL((GVL_XTS.StationCtrl[nStationSelected].eCmd = E_STATION_CTRL.STATION_ENABLE),        FALSE, TRUE);
bStationEnter                         := SEL((GVL_XTS.StationCtrl[nStationSelected].eCmd = E_STATION_CTRL.STATION_MOVER_ENTER),   FALSE, TRUE);
bStationStart                         := SEL((GVL_XTS.StationCtrl[nStationSelected].eCmd = E_STATION_CTRL.STATION_PROCESS_START), FALSE, TRUE);
bStationDone                          := SEL((GVL_XTS.StationCtrl[nStationSelected].eCmd = E_STATION_CTRL.STATION_PROCESS_DONE),  FALSE, TRUE);
bStationOut                           := SEL((GVL_XTS.StationCtrl[nStationSelected].eCmd = E_STATION_CTRL.STATION_MOVER_OUT),     FALSE, TRUE);
bStationGone                          := SEL((GVL_XTS.StationCtrl[nStationSelected].eCmd = E_STATION_CTRL.STATION_MOVER_GONE),    FALSE, TRUE);

eMoverState                           := f_GetState   (GVL_XTS.MoverState[nMoverSelected].State);
eMoverResult                          := f_GetProgress(GVL_XTS.MoverState[nMoverSelected].State);

sMoverState                           := TO_STRING(eMoverState);
sMoverResult                          := TO_STRING(eMoverResult);

sStationState                         := TO_STRING(GVL_XTS.StationState[nStationSelected].eState);
sStationStateMask                     := Tc2_Utilities.BYTE_TO_BINSTR(GVL_XTS.StationState[nStationSelected].nMask, 8);
sStationCtrlMask                      := Tc2_Utilities.BYTE_TO_BINSTR(GVL_XTS.StationCtrl[nStationSelected].nMask, 8);

tStationSelectedQueue                 := GVL_XTS.StationQueue[nStationSelected];

ACTION StationParameterInit:
//---------------------------------------------------------------------------------------
//---------------------------------------------------------------------------------------
//
//
//---------------------------------------------------------------------------------------
//---------------------------------------------------------------------------------------
nStn                    := 1;
GVL_XTS.StationParameter[nStn].sText               := 'STN_12';
GVL_XTS.StationParameter[nStn].rPosWait            :=   6250.0; // absolute modulo position
GVL_XTS.StationParameter[nStn].rPosStop[1]         :=     62.5; // relative to rPosWait
GVL_XTS.StationParameter[nStn].rReleaseDistance    :=     -5.0; // relative to Mover.ActPos

GVL_XTS.StationParameter[nStn].rGap                :=    105.0;
GVL_XTS.StationParameter[nStn].rVelo               :=   1750.0;
GVL_XTS.StationParameter[nStn].rAccDec             :=  17500.0;
GVL_XTS.StationParameter[nStn].rJerk               := 800000.0;
//---------------------------------------------------------------------------------------
//---------------------------------------------------------------------------------------
//
//
//---------------------------------------------------------------------------------------
//---------------------------------------------------------------------------------------
nStn                    := 2;
GVL_XTS.StationParameter[nStn].sText               := 'STN_01(1)';
GVL_XTS.StationParameter[nStn].rPosWait            :=    125.0; // absolute modulo position
GVL_XTS.StationParameter[nStn].rPosStop[1]         :=     62.5; // relative to rPosWait
GVL_XTS.StationParameter[nStn].rReleaseDistance    :=     40.0; // relative to Mover.ActPos

GVL_XTS.StationParameter[nStn].rGap                :=    105.0;
GVL_XTS.StationParameter[nStn].rVelo               :=   2500.0;
GVL_XTS.StationParameter[nStn].rAccDec             :=  17500.0;
GVL_XTS.StationParameter[nStn].rJerk               := 800000.0;

nStn                    := 3;
GVL_XTS.StationParameter[nStn].sText               := 'STN_01(2)';
GVL_XTS.StationParameter[nStn].rPosWait            :=    125.0; // absolute modulo position
GVL_XTS.StationParameter[nStn].rPosStop[1]         :=    187.5; // relative to rPosWait
GVL_XTS.StationParameter[nStn].rReleaseDistance    :=     30.0; // relative to Mover.ActPos

GVL_XTS.StationParameter[nStn].rGap                :=    105.0;
GVL_XTS.StationParameter[nStn].rVelo               :=   2500.0;
GVL_XTS.StationParameter[nStn].rAccDec             :=  17500.0;
GVL_XTS.StationParameter[nStn].rJerk               := 800000.0;

nStn                    := 4;
GVL_XTS.StationParameter[nStn].sText               := 'STN_01(3)';
GVL_XTS.StationParameter[nStn].rPosWait            :=    125.0; // absolute modulo position
GVL_XTS.StationParameter[nStn].rPosStop[1]         :=    312.5; // relative to rPosWait
GVL_XTS.StationParameter[nStn].rReleaseDistance    :=     20.0; // relative to Mover.ActPos

GVL_XTS.StationParameter[nStn].rGap                :=    105.0;
GVL_XTS.StationParameter[nStn].rVelo               :=   2500.0;
GVL_XTS.StationParameter[nStn].rAccDec             :=  17500.0;
GVL_XTS.StationParameter[nStn].rJerk               := 800000.0;

nStn                    := 5;
GVL_XTS.StationParameter[nStn].sText               := 'STN_01(4)';
GVL_XTS.StationParameter[nStn].rPosWait            :=    125.0; // absolute modulo position
GVL_XTS.StationParameter[nStn].rPosStop[1]         :=    437.5; // relative to rPosWait
GVL_XTS.StationParameter[nStn].rReleaseDistance    :=     10.0; // relative to Mover.ActPos

GVL_XTS.StationParameter[nStn].rGap                :=    105.0;
GVL_XTS.StationParameter[nStn].rVelo               :=   2500.0;
GVL_XTS.StationParameter[nStn].rAccDec             :=  17500.0;
GVL_XTS.StationParameter[nStn].rJerk               := 800000.0;
//---------------------------------------------------------------------------------------
//---------------------------------------------------------------------------------------
//
//
//---------------------------------------------------------------------------------------
//---------------------------------------------------------------------------------------
nStn                    := 6;
GVL_XTS.StationParameter[nStn].sText               := 'STN_02(1)';
GVL_XTS.StationParameter[nStn].rPosWait            :=   1140.0; // absolute modulo position

GVL_XTS.StationParameter[nStn].nConfiguredStopCount:=      2;
GVL_XTS.StationParameter[nStn].rPosStop[1]         :=    162.5; // relative to rPosWait
GVL_XTS.StationParameter[nStn].rPosStop[2]         :=    202.5; // relative to rPosWait

GVL_XTS.StationParameter[nStn].rReleaseDistance    :=    150.0; // relative to Mover.ActPos

GVL_XTS.StationParameter[nStn].rGap                :=    105.0;
GVL_XTS.StationParameter[nStn].rVelo               :=   2500.0;
GVL_XTS.StationParameter[nStn].rAccDec             :=  17500.0;
GVL_XTS.StationParameter[nStn].rJerk               := 800000.0;


nStn                    := 7;
GVL_XTS.StationParameter[nStn].sText               := 'STN_02(2)';
GVL_XTS.StationParameter[nStn].rPosWait            :=   1140.0; // absolute modulo position

GVL_XTS.StationParameter[nStn].nConfiguredStopCount:=      2;
GVL_XTS.StationParameter[nStn].rPosStop[1]         :=    268.5; // relative to rPosWait
GVL_XTS.StationParameter[nStn].rPosStop[2]         :=    307.5; // relative to rPosWait

GVL_XTS.StationParameter[nStn].rReleaseDistance    :=    100.0; // relative to Mover.ActPos

GVL_XTS.StationParameter[nStn].rGap                :=    105.0;
GVL_XTS.StationParameter[nStn].rVelo               :=   2500.0;
GVL_XTS.StationParameter[nStn].rAccDec             :=  17500.0;
GVL_XTS.StationParameter[nStn].rJerk               := 800000.0;
//---------------------------------------------------------------------------------------
//---------------------------------------------------------------------------------------
//---------------------------------------------------------------------------------------
//---------------------------------------------------------------------------------------
//
//
//---------------------------------------------------------------------------------------
//---------------------------------------------------------------------------------------
nStn                    := 8;
GVL_XTS.StationParameter[nStn].sText               := 'STN_03';
GVL_XTS.StationParameter[nStn].rPosWait            :=   1675.0; // absolute modulo position
GVL_XTS.StationParameter[nStn].rPosStop[1]         :=     60.5; // relative to rPosWait
GVL_XTS.StationParameter[nStn].rReleaseDistance    :=      2.0; // relative to Mover.ActPos

GVL_XTS.StationParameter[nStn].rGap                :=    105.0;
GVL_XTS.StationParameter[nStn].rVelo               :=    500.0;
GVL_XTS.StationParameter[nStn].rAccDec             :=  17500.0;
GVL_XTS.StationParameter[nStn].rJerk               := 800000.0;
//---------------------------------------------------------------------------------------
//---------------------------------------------------------------------------------------
//---------------------------------------------------------------------------------------
//---------------------------------------------------------------------------------------
//
//
//---------------------------------------------------------------------------------------
//---------------------------------------------------------------------------------------
nStn                    := 9;
GVL_XTS.StationParameter[nStn].sText               := 'STN_04';
GVL_XTS.StationParameter[nStn].rPosWait            :=   2000.0; // absolute modulo position

GVL_XTS.StationParameter[nStn].nConfiguredStopCount:=      2;
GVL_XTS.StationParameter[nStn].rPosStop[1]         :=    187.5; // relative to rPosWait
GVL_XTS.StationParameter[nStn].rPosStop[2]         :=    125.0; // relative to rPosWait

GVL_XTS.StationParameter[nStn].rReleaseDistance    :=     62.5; // relative to Mover.ActPos

GVL_XTS.StationParameter[nStn].rGap                :=    105.0;
GVL_XTS.StationParameter[nStn].rVelo               :=   2500.0;
GVL_XTS.StationParameter[nStn].rAccDec             :=  17500.0;
GVL_XTS.StationParameter[nStn].rJerk               := 800000.0;
//---------------------------------------------------------------------------------------
//---------------------------------------------------------------------------------------
//---------------------------------------------------------------------------------------
//---------------------------------------------------------------------------------------
//
//
//---------------------------------------------------------------------------------------
//---------------------------------------------------------------------------------------
nStn                    := 10;
GVL_XTS.StationParameter[nStn].sText               := 'STN_05';
GVL_XTS.StationParameter[nStn].rPosWait            :=   2000.0; // absolute modulo position

GVL_XTS.StationParameter[nStn].nConfiguredStopCount:=      2;
GVL_XTS.StationParameter[nStn].rPosStop[1]         :=    462.5; // relative to rPosWait
GVL_XTS.StationParameter[nStn].rPosStop[2]         :=    400.0; // relative to rPosWait

GVL_XTS.StationParameter[nStn].rReleaseDistance    :=     10.0; // relative to Mover.ActPos

GVL_XTS.StationParameter[nStn].rGap                :=    105.0;
GVL_XTS.StationParameter[nStn].rVelo               :=   2500.0;
GVL_XTS.StationParameter[nStn].rAccDec             :=  17500.0;
GVL_XTS.StationParameter[nStn].rJerk               := 800000.0;
//---------------------------------------------------------------------------------------
//---------------------------------------------------------------------------------------
//---------------------------------------------------------------------------------------
//---------------------------------------------------------------------------------------
//
//
//---------------------------------------------------------------------------------------
//---------------------------------------------------------------------------------------
nStn                    := 11;
GVL_XTS.StationParameter[nStn].sText               := 'STN_06(1)';
GVL_XTS.StationParameter[nStn].rPosWait            :=   3000.0; // absolute modulo position
GVL_XTS.StationParameter[nStn].rPosStop[1]         :=     62.5; // relative to rPosWait
GVL_XTS.StationParameter[nStn].rReleaseDistance    :=     40.0; // relative to Mover.ActPos

GVL_XTS.StationParameter[nStn].rGap                :=    105.0;
GVL_XTS.StationParameter[nStn].rVelo               :=   2500.0;
GVL_XTS.StationParameter[nStn].rAccDec             :=  17500.0;
GVL_XTS.StationParameter[nStn].rJerk               := 800000.0;

nStn                    := 12;
GVL_XTS.StationParameter[nStn].sText               := 'STN_06(2)';
GVL_XTS.StationParameter[nStn].rPosWait            :=   3000.0; // absolute modulo position
GVL_XTS.StationParameter[nStn].rPosStop[1]         :=    187.5; // relative to rPosWait
GVL_XTS.StationParameter[nStn].rReleaseDistance    :=     30.0; // relative to Mover.ActPos

GVL_XTS.StationParameter[nStn].rGap                :=    105.0;
GVL_XTS.StationParameter[nStn].rVelo               :=   2500.0;
GVL_XTS.StationParameter[nStn].rAccDec             :=  17500.0;
GVL_XTS.StationParameter[nStn].rJerk               := 800000.0;

nStn                    := 13;
GVL_XTS.StationParameter[nStn].sText               := 'STN_06(3)';
GVL_XTS.StationParameter[nStn].rPosWait            :=   3000.0; // absolute modulo position
GVL_XTS.StationParameter[nStn].rPosStop[1]         :=    312.5; // relative to rPosWait
GVL_XTS.StationParameter[nStn].rReleaseDistance    :=     20.0; // relative to Mover.ActPos

GVL_XTS.StationParameter[nStn].rGap                :=    105.0;
GVL_XTS.StationParameter[nStn].rVelo               :=   2500.0;
GVL_XTS.StationParameter[nStn].rAccDec             :=  17500.0;
GVL_XTS.StationParameter[nStn].rJerk               := 800000.0;

nStn                    := 14;
GVL_XTS.StationParameter[nStn].sText               := 'STN_06(4)';
GVL_XTS.StationParameter[nStn].rPosWait            :=   3000.0; // absolute modulo position
GVL_XTS.StationParameter[nStn].rPosStop[1]         :=    437.5; // relative to rPosWait
GVL_XTS.StationParameter[nStn].rReleaseDistance    :=     10.0; // relative to Mover.ActPos

GVL_XTS.StationParameter[nStn].rGap                :=    105.0;
GVL_XTS.StationParameter[nStn].rVelo               :=   2500.0;
GVL_XTS.StationParameter[nStn].rAccDec             :=  17500.0;
GVL_XTS.StationParameter[nStn].rJerk               := 800000.0;
//---------------------------------------------------------------------------------------
//---------------------------------------------------------------------------------------
//---------------------------------------------------------------------------------------
//---------------------------------------------------------------------------------------
//
//
//---------------------------------------------------------------------------------------
//---------------------------------------------------------------------------------------
nStn                    := 15;
GVL_XTS.StationParameter[nStn].sText               := 'STN_07';
GVL_XTS.StationParameter[nStn].rPosWait            :=   4000.0; // absolute modulo position

GVL_XTS.StationParameter[nStn].nConfiguredStopCount:=      2;
GVL_XTS.StationParameter[nStn].rPosStop[1]         :=     62.5; // relative to rPosWait
GVL_XTS.StationParameter[nStn].rPosStop[2]         :=    102.5; // relative to rPosWait

GVL_XTS.StationParameter[nStn].rReleaseDistance    :=     10.0; // relative to Mover.ActPos

GVL_XTS.StationParameter[nStn].rGap                :=    105.0;
GVL_XTS.StationParameter[nStn].rVelo               :=   2500.0;
GVL_XTS.StationParameter[nStn].rAccDec             :=  17500.0;
GVL_XTS.StationParameter[nStn].rJerk               := 800000.0;
//---------------------------------------------------------------------------------------
//---------------------------------------------------------------------------------------
//---------------------------------------------------------------------------------------
//---------------------------------------------------------------------------------------
//
//
//---------------------------------------------------------------------------------------
//---------------------------------------------------------------------------------------
nStn                    := 16;
GVL_XTS.StationParameter[nStn].sText               := 'STN_08';
GVL_XTS.StationParameter[nStn].rPosWait            :=   4250.0; // absolute modulo position
GVL_XTS.StationParameter[nStn].rPosStop[1]         :=     62.5; // relative to rPosWait
GVL_XTS.StationParameter[nStn].rReleaseDistance    :=     10.0; // relative to Mover.ActPos

GVL_XTS.StationParameter[nStn].rGap                :=    105.0;
GVL_XTS.StationParameter[nStn].rVelo               :=   2500.0;
GVL_XTS.StationParameter[nStn].rAccDec             :=  17500.0;
GVL_XTS.StationParameter[nStn].rJerk               := 800000.0;
//---------------------------------------------------------------------------------------
//---------------------------------------------------------------------------------------
//---------------------------------------------------------------------------------------
//---------------------------------------------------------------------------------------
//
//
//---------------------------------------------------------------------------------------
//---------------------------------------------------------------------------------------
nStn                    := 17;
GVL_XTS.StationParameter[nStn].sText               := 'STN_09';
GVL_XTS.StationParameter[nStn].rPosWait            :=   4500.0; // absolute modulo position
GVL_XTS.StationParameter[nStn].rPosStop[1]         :=     62.5; // relative to rPosWait
GVL_XTS.StationParameter[nStn].rReleaseDistance    :=    125.0; // relative to Mover.ActPos

GVL_XTS.StationParameter[nStn].rGap                :=    105.0;
GVL_XTS.StationParameter[nStn].rVelo               :=   2500.0;
GVL_XTS.StationParameter[nStn].rAccDec             :=  17500.0;
GVL_XTS.StationParameter[nStn].rJerk               := 800000.0;
//---------------------------------------------------------------------------------------
//---------------------------------------------------------------------------------------
//---------------------------------------------------------------------------------------
//---------------------------------------------------------------------------------------
//
//
//---------------------------------------------------------------------------------------
//---------------------------------------------------------------------------------------
nStn                    := 18;
GVL_XTS.StationParameter[nStn].sText               := 'STN_10';
GVL_XTS.StationParameter[nStn].rPosWait            :=   4875.0; // absolute modulo position
GVL_XTS.StationParameter[nStn].rPosStop[1]         :=     60.0; // relative to rPosWait
GVL_XTS.StationParameter[nStn].rReleaseDistance    :=     2.5; // relative to Mover.ActPos

GVL_XTS.StationParameter[nStn].rGap                :=    105.0;
GVL_XTS.StationParameter[nStn].rVelo               :=    500.0;
GVL_XTS.StationParameter[nStn].rAccDec             :=  17500.0;
GVL_XTS.StationParameter[nStn].rJerk               := 800000.0;
//---------------------------------------------------------------------------------------
//---------------------------------------------------------------------------------------
//---------------------------------------------------------------------------------------
//---------------------------------------------------------------------------------------
//
//
//---------------------------------------------------------------------------------------
//---------------------------------------------------------------------------------------
nStn                    := 19;
GVL_XTS.StationParameter[nStn].sText               := 'STN_11(1)';
GVL_XTS.StationParameter[nStn].rPosWait            :=   5250.0; // absolute modulo position
GVL_XTS.StationParameter[nStn].rPosStop[1]         :=     62.5; // relative to rPosWait
GVL_XTS.StationParameter[nStn].rReleaseDistance    :=    110.0; // relative to Mover.ActPos

GVL_XTS.StationParameter[nStn].rGap                :=    105.0;
GVL_XTS.StationParameter[nStn].rVelo               :=   2500.0;
GVL_XTS.StationParameter[nStn].rAccDec             :=  17500.0;
GVL_XTS.StationParameter[nStn].rJerk               := 800000.0;

nStn                    := 20;
GVL_XTS.StationParameter[nStn].sText               := 'STN_11(2)';
GVL_XTS.StationParameter[nStn].rPosWait            :=   5250.0; // absolute modulo position
GVL_XTS.StationParameter[nStn].rPosStop[1]         :=    187.5; // relative to rPosWait
GVL_XTS.StationParameter[nStn].rReleaseDistance    :=    100.0; // relative to Mover.ActPos

GVL_XTS.StationParameter[nStn].rGap                :=    105.0;
GVL_XTS.StationParameter[nStn].rVelo               :=   2500.0;
GVL_XTS.StationParameter[nStn].rAccDec             :=  17500.0;
GVL_XTS.StationParameter[nStn].rJerk               := 800000.0;

nStn                    := 21;
GVL_XTS.StationParameter[nStn].sText               := 'STN_11(3)';
GVL_XTS.StationParameter[nStn].rPosWait            :=   5250.0; // absolute modulo position
GVL_XTS.StationParameter[nStn].rPosStop[1]         :=    312.5; // relative to rPosWait
GVL_XTS.StationParameter[nStn].rReleaseDistance    :=     90.0; // relative to Mover.ActPos

GVL_XTS.StationParameter[nStn].rGap                :=    105.0;
GVL_XTS.StationParameter[nStn].rVelo               :=   2500.0;
GVL_XTS.StationParameter[nStn].rAccDec             :=  17500.0;
GVL_XTS.StationParameter[nStn].rJerk               := 800000.0;

nStn                    := 22;
GVL_XTS.StationParameter[nStn].sText               := 'STN_11(4)';
GVL_XTS.StationParameter[nStn].rPosWait            :=   5250.0; // absolute modulo position
GVL_XTS.StationParameter[nStn].rPosStop[1]         :=    437.5; // relative to rPosWait
GVL_XTS.StationParameter[nStn].rReleaseDistance    :=     80.0; // relative to Mover.ActPos

GVL_XTS.StationParameter[nStn].rGap                :=    105.0;
GVL_XTS.StationParameter[nStn].rVelo               :=   2500.0;
GVL_XTS.StationParameter[nStn].rAccDec             :=  17500.0;
GVL_XTS.StationParameter[nStn].rJerk               := 800000.0;
//---------------------------------------------------------------------------------------
//---------------------------------------------------------------------------------------
END_ACTION

END_PROGRAM

// ---- MSG/MessageData.TcPOU
PROGRAM MessageData
VAR CONSTANT
{attribute 'hide'}
  STR_LEN       : UINT := 65535;
END_VAR
VAR_INPUT
	bPowerFail		: BOOL;   // UPS switch
	bWriteFile		: BOOL;   // manual write of list
	bReset				: BOOL;
	pList					: POINTER TO ARRAY[1..GVL_MSG.MAX_MESSAGE] OF ST_Message; // attach your list here
	pLocalTime		: POINTER TO DT; 
END_VAR
VAR_OUTPUT
	bBusy					: BOOL;
  bDone         : BOOL;
	VisuList		  : ARRAY[1..GVL_MSG.MAX_MESSAGE] OF ST_Message;
END_VAR
VAR
	eState 				: E_MESSAGE_STATE;

	rtrigReset		: Tc2_Standard.R_TRIG;
	aWriteList		: ARRAY[1..GVL_MSG.MAX_MESSAGE] OF ST_Message;
	sWriteData		: STRING(STR_LEN);
	sNewLine			: STRING := '$N';
	sTab					: STRING := '$T';
	iCount, 
	iStart, 
	iEnd					: UINT;

	fbCreateDir		: Tc2_System.FB_CreateDir;
	sTmp          : STRING(256);
	sFilename			: STRING(256);
	sFolderDate		: STRING;
	bFileCreated	: BOOL;

	fbFileOpen		  : Tc2_System.FB_FileOpen;
	fbFileWrite		  : Tc2_System.FB_FileWrite;
	fbFileClose		  : Tc2_System.FB_FileClose;

  ivis          : UINT;

  bBusyWrite,
  bErrorWrite   : BOOL;
  nErrorWrite   : UDINT;
  nStateWrite   : UINT;
END_VAR

//-----------------------------------------------------------------------------
// check pointers
//-----------------------------------------------------------------------------
IF NOT (pList <> 0) OR
   NOT (pLocalTime <> 0)
THEN
  eState                      := MSG_INVALID_POINTERS;
  RETURN;
END_IF
//-----------------------------------------------------------------------------
// check date
// new message file for a new day
//-----------------------------------------------------------------------------
IF (FolderDate(pLocalTime) <> sFolderDate)
THEN
  bFileCreated                := FALSE;
END_IF
//-----------------------------------------------------------------------------
//----------------------------------------------------------------------------- 
rtrigReset(CLK:= bReset);
IF rtrigReset.Q
THEN
  bReset                      := FALSE;
  eState                      := MSG_NULL;
END_IF
//-----------------------------------------------------------------------------
//-----------------------------------------------------------------------------
CASE eState OF
  MSG_NULL:
    bBusy                     := 
    bDone                     := FALSE;

    IF (GVL_MSG.MessageIndex > GVL_MSG.MAX_MESSAGE/2)
    THEN
      eState                  := MSG_INIT;

    ELSIF (bWriteFile) OR (bPowerFail)
    THEN
      eState                  := MSG_INIT;

      IF (GVL_MSG.MessageIndex = 0)
      THEN
        bBusy                 := TRUE;
        eState                := MSG_WRITE_FILE_DONE;
      END_IF
    END_IF
END_CASE
//-----------------------------------------------------------------------------
CASE eState OF
  MSG_INIT:
    WriteData(FALSE);

    // clear intern list
    memset(ADR(aWriteList),     0, SIZEOF(aWriteList));

    // copy from attached list to local
    memcpy(ADR(aWriteList), pList, SIZEOF(aWriteList));

    // clear attached list
    memset(pList, 0, SIZEOF(aWriteList));

    bBusy                     := TRUE;
    iStart 	                  := 1;
    iEnd 		                  := SEL((GVL_MSG.MessageIndex > GVL_MSG.MAX_MESSAGE-1),
                                      GVL_MSG.MessageIndex,
                                      GVL_MSG.MAX_MESSAGE);
    GVL_MSG.MessageIndex      := 0;

    IF NOT bFileCreated
    THEN
      // folder and filename have to be created
      eState                  := MSG_ROOT;
    ELSE
      // folder and file already exist
      eState                  := MSG_LINE_START;
    END_IF
END_CASE
//-----------------------------------------------------------------------------
CASE eState OF
  MSG_ROOT:
    eState                    := MSG_ROOT_CREATE;
    fbCreateDir.sPathName     := left(GVL_MSG.LOG_DIR,len(GVL_MSG.LOG_DIR)-1);
    fbCreateDir(
            bExecute	        := FALSE);
  
  MSG_ROOT_CREATE:
    (* create root folder *)
    fbCreateDir(
            bExecute	        := TRUE);
    IF fbCreateDir.bBusy
    THEN
      eState                  := MSG_ROOT_CREATE_BUSY;
    END_IF
  
  MSG_ROOT_CREATE_BUSY:
    fbCreateDir(
            bExecute	        := TRUE);
    IF NOT fbCreateDir.bBusy
    THEN
      eState                  := MSG_FOLDER;
    END_IF
  
  MSG_FOLDER:
    eState                    := MSG_FOLDER_CREATE;
    sFolderDate               := FolderDate(pLocalTime);
    fbCreateDir.sPathName     := concat(GVL_MSG.LOG_DIR, sFolderDate);
    fbCreateDir(
            bExecute	        := FALSE);

  MSG_FOLDER_CREATE:
    (* create active folder *)
    fbCreateDir(
            bExecute	        := TRUE);
    IF fbCreateDir.bBusy
    THEN
      eState                  := MSG_FOLDER_CREATE_BUSY;
    END_IF
  
  MSG_FOLDER_CREATE_BUSY:
    fbCreateDir(
            bExecute	        := TRUE);
    IF NOT fbCreateDir.bBusy
    THEN
      eState                  := MSG_FILE_CREATE_DONE;
      fbCreateDir(
              bExecute	      := FALSE);
    END_IF
END_CASE
//-----------------------------------------------------------------------------
CASE eState OF
  MSG_FILE_CREATE_DONE:
    eState                    := MSG_LINE_START;
    bFileCreated              := TRUE;
    // build complete file path
    sTmp                      := concat(concat(GVL_MSG.LOG_FILE, sFolderDate),'.txt');
    sTmp                      := concat('\', sTmp);
    sFilename                 := concat(fbCreateDir.sPathName, sTmp);
END_CASE
//-----------------------------------------------------------------------------
CASE eState OF
  MSG_LINE_START:
    GVL_MSG.MessageError      := 0;
    eState                    := MSG_LINE_BUILD;
    iCount                    := iStart;
    memset(ADR(sWriteData),0,SIZEOF(sWriteData));
END_CASE
//-----------------------------------------------------------------------------
CASE eState OF
  MSG_LINE_BUILD:
    eState                    := MSG_LINE_CHECK;
    IF (aWriteList[iCount].eType > E_MessageType.eMessageEmpty)
    THEN
      sTmp                    := TO_STRING(aWriteList[iCount].eType);
      sTmp                    := Tc2_Standard.CONCAT(sTmp, sTab);
      sTmp                    := Tc2_Standard.CONCAT(sTmp, aWriteList[iCount].tTime);
      sTmp                    := Tc2_Standard.CONCAT(sTmp, sTab);
      sTmp                    := Tc2_Standard.CONCAT(sTmp, Device_To_String(aWriteList[iCount].eDevice));
      sTmp                    := Tc2_Standard.CONCAT(sTmp, sTab);
      sTmp                    := Tc2_Standard.CONCAT(sTmp, TO_STRING(aWriteList[iCount].eSubdevice));
      sTmp                    := Tc2_Standard.CONCAT(sTmp, sTab);
      sTmp                    := Tc2_Standard.CONCAT(sTmp, TO_STRING(aWriteList[iCount].iErrorNumber));
      sTmp                    := Tc2_Standard.CONCAT(sTmp, sTab);
      sTmp                    := Tc2_Standard.CONCAT(sTmp, aWriteList[iCount].sText);
      sTmp                    := Tc2_Standard.CONCAT(sTmp, sNewLine);
      Builder(ADR(sTmp), ADR(sWriteData), StringLen(ADR(sTmp)));
    END_IF
    iCount                    := iCount + 1;
END_CASE
//-----------------------------------------------------------------------------
CASE eState OF
  MSG_LINE_CHECK:
  IF NOT (iCount > iEnd)
  THEN
    eState                    := MSG_LINE_BUILD;
  ELSE
    IF (StringLen(ADR(sWriteData)) > 1)
    THEN
      eState                  := MSG_WRITE_FILE_BUSY;
    ELSE
      eState                  := MSG_WRITE_FILE_DONE;
    END_IF
  END_IF
  
  MSG_WRITE_FILE_BUSY:
  IF WriteData(TRUE)
  THEN
    eState                    := MSG_WRITE_FILE_END;
  END_IF
  
  MSG_WRITE_FILE_END:
  WriteData(FALSE);
  eState                      := MSG_WRITE_FILE_DONE;
  
  MSG_WRITE_FILE_DONE:
  bDone                       := TRUE;
  IF NOT (bWriteFile)
  THEN
    eState                    := MSG_NULL;
  END_IF
END_CASE
//-----------------------------------------------------------------------------
//-----------------------------------------------------------------------------
// visu message list
//-----------------------------------------------------------------------------
memset(ADR(VisuList),0,SIZEOF(VisuList));
// copy last written message list to visu message list
memcpy(ADR(VisuList), ADR(aWriteList), SIZEOF(VisuList));
//-----------------------------------------------------------------------------

METHOD Builder : BOOL // string concat for length > 255
VAR_INPUT
  pInString   : POINTER TO STRING;
  pOutString  : POINTER TO STRING(STR_LEN);
  Length      : UINT;
END_VAR
VAR
  Counter     : DINT;
  pInWork     : POINTER TO BYTE;
  pOutWork    : POINTER TO BYTE;
END_VAR
pOutWork := pOutString;
pInWork := pInString;
Counter := 0;

(*check termination*)
WHILE (pOutWork^ <> 0) AND
      (Counter < STR_LEN+1)
DO
  Counter := Counter + 1;
  pOutWork := pOutWork + 1;
END_WHILE

(* append only if data fits into output *)
IF (Counter + Length < STR_LEN+1)
THEN

  (* append data *)
  FOR Counter := 1 TO Length
  DO
    pOutWork^ := pInWork^;
    pOutWork := pOutWork + 1;
    pInWork := pInWork + 1;
  END_FOR

  (* terminate *)
  pOutWork := pOutWork + 1;
  pOutWork^ := 0;
END_IF
END_METHOD

METHOD Device_to_String : string
VAR_INPUT
  eMsgDevice    : e_Device;
END_VAR
VAR
  sId                 : STRING := '_ID_';
  nId                 : UDINT;
END_VAR
IF (eMsgDevice <= e_device.General)
THEN
  // general case with no added indices
  Device_to_String := TO_STRING(eMsgDevice);
ELSE
  IF (eMsgDevice >= e_Device.Process)
  THEN
    nId := eMsgDevice MOD e_Device.Process;
    sId := concat(sId, TO_STRING(nId));
 
    Device_to_String := concat(TO_STRING(e_Device.Process), sId);

  ELSIF (eMsgDevice >= e_Device.Data)
  THEN
    nId := eMsgDevice MOD e_Device.Data;
    sId := concat(sId, TO_STRING(nId));
 
    Device_to_String := concat(TO_STRING(e_device.Data), sId);

  ELSIF (eMsgDevice >= e_device.XfcAxis)
  THEN
    nId := eMsgDevice MOD e_device.XfcAxis;
    sId := concat(sId, TO_STRING(nId));
 
    Device_to_String := concat(TO_STRING(e_device.XfcAxis), sId);

  ELSIF (eMsgDevice >= e_device.Axis)
  THEN
    nId := eMsgDevice MOD e_device.Axis;
    sId := concat(sId, TO_STRING(nId));
 
    Device_to_String := concat(TO_STRING(e_device.Axis), sId);

  ELSIF (eMsgDevice >= e_device.NciChannelCtrl)
  THEN
    nId := eMsgDevice MOD e_device.NciChannelCtrl;
    sId := concat(sId, TO_STRING(nId));
 
    Device_to_String := concat(TO_STRING(e_device.NciChannelCtrl), sId);

  ELSIF (eMsgDevice >= e_device.NciChannel)
  THEN
    nId := eMsgDevice MOD e_device.NciChannel;
    sId := concat(sId, TO_STRING(nId));
 
    Device_to_String := concat(TO_STRING(e_device.NciChannel), sId);

  ELSIF (eMsgDevice >= e_Device.Camming)
  THEN
    nId := eMsgDevice MOD e_Device.Camming;
    sId := concat(sId, TO_STRING(nId));
 
    Device_to_String := concat(TO_STRING(e_device.Camming), sId);

  ELSIF (eMsgDevice >= e_Device.XtsStation)
  THEN
    nId := eMsgDevice MOD e_Device.XtsStation;
    sId := concat(sId, TO_STRING(nId));
 
    Device_to_String := concat(TO_STRING(e_device.XtsStation), sId);

  ELSIF (eMsgDevice >= e_Device.XfcTouchProbe)
  THEN
    nId := eMsgDevice MOD e_Device.XfcTouchProbe;
    sId := concat(sId, TO_STRING(nId));
 
    Device_to_String := concat(TO_STRING(e_device.XfcTouchProbe), sId);

  ELSIF (eMsgDevice >= e_Device.XfcTriggerBox)
  THEN
    nId := eMsgDevice MOD e_Device.XfcTriggerBox;
    sId := concat(sId, TO_STRING(nId));
 
    Device_to_String := concat(TO_STRING(e_device.XfcTriggerBox), sId);

  ELSIF (eMsgDevice >= e_Device.XtsTransportUnit)
  THEN
    nId := eMsgDevice MOD e_Device.XtsTransportUnit;
    sId := concat(sId, TO_STRING(nId));
 
    Device_to_String := concat(TO_STRING(e_device.XtsTransportUnit), sId);

  ELSIF (eMsgDevice >= e_Device.MoverCtrl)
  THEN
    nId := eMsgDevice MOD e_Device.MoverCtrl;
    sId := concat(sId, TO_STRING(nId));
 
    Device_to_String := concat(TO_STRING(e_device.MoverCtrl), sId);

  ELSIF (eMsgDevice >= e_Device.Mover)
  THEN
    nId := eMsgDevice MOD e_Device.Mover;
    sId := concat(sId, TO_STRING(nId));
 
    Device_to_String := concat(TO_STRING(e_device.Mover), sId);

  ELSIF (eMsgDevice >= e_Device.XpuCtrl)
  THEN
    nId := eMsgDevice MOD e_Device.XpuCtrl;
    sId := concat(sId, TO_STRING(nId));
 
    Device_to_String := concat(TO_STRING(e_device.XpuCtrl), sId);

  ELSIF (eMsgDevice >= e_Device.Xpu)
  THEN
    nId := eMsgDevice MOD e_Device.Xpu;
    sId := concat(sId, TO_STRING(nId));
 
    Device_to_String := concat(TO_STRING(e_device.Xpu), sId);

  ELSIF (eMsgDevice >= e_Device.CaGroup)
  THEN
    nId := eMsgDevice MOD e_Device.CaGroup;
    sId := concat(sId, TO_STRING(nId));
 
    Device_to_String := concat(TO_STRING(e_device.CaGroup), sId);

  ELSE
    Device_to_String := TO_STRING(eMsgDevice);
  END_IF
END_IF
END_METHOD

METHOD FolderDate : STRING
VAR_INPUT
	pLocalTime		: POINTER TO DT;
END_VAR
VAR
	sTmp					: STRING;
END_VAR
IF NOT (pLocalTime <> 0)
THEN
	FolderDate := 'NULL';
	RETURN;
END_IF

sTmp := DT_TO_STRING(pLocalTime^);

// cut off #dt literal
sTmp := right(sTmp, len(sTmp)-3);

sTmp := replace(sTmp, '_', 1, 5);
sTmp := replace(sTmp, '_', 1, 8);

sTmp := left(sTmp,10);	// year_month_day

FolderDate := sTmp;
END_METHOD

METHOD StringLen : UINT // 	string length for len > 255
VAR_INPUT
  pInString		: POINTER TO STRING(32767);
END_VAR
VAR
	Counter			: UINT;
	pInWork			: POINTER TO BYTE;
END_VAR
pInWork := pInString;
Counter := 0;

WHILE (pInWork^ <> 0) AND
			(Counter < 32767)
DO
	Counter := Counter + 1;
	pInWork := pInWork + 1;
END_WHILE

StringLen := Counter;
END_METHOD

METHOD WriteData  : BOOL
VAR_INPUT
  bExecute        : BOOL;
END_VAR
VAR
END_VAR

IF NOT bExecute
THEN
  bBusyWrite                := FALSE;
	nStateWrite               := 0;
END_IF

CASE nStateWrite OF

	0:
		fbFileOpen.bExecute		  := FALSE;
		fbFileWrite.bExecute	  := FALSE;
		fbFileClose.bExecute	  := FALSE;

		IF bExecute
		THEN
			bBusyWrite            := TRUE;
			nStateWrite           := 10;
		END_IF

	10:
		fbFileOpen.bExecute     := TRUE;
		IF fbFileOpen.bBusy
		THEN
			nStateWrite           := 20;
		END_IF

	20:
		IF NOT fbFileOpen.bBusy
		THEN
			fbFileOpen.bExecute   := FALSE;
			fbFileWrite.bExecute  := TRUE;
			nStateWrite           := 30;
		END_IF

	30:
		IF fbFileWrite.bBusy
		THEN
			nStateWrite           := 40;
		END_IF

	40:
		IF NOT fbFileWrite.bBusy
		THEN
			fbFileWrite.bExecute  := FALSE;
			fbFileClose.bExecute  := TRUE;
			nStateWrite           := 50;
		END_IF

	50:
		IF fbFileClose.bBusy
		THEN
			nStateWrite           := 60;
		END_IF

	60:
		IF NOT fbFileClose.bBusy
		THEN
			fbFileClose.bExecute  := FALSE;
			nStateWrite 		      := 100;
		END_IF
	
	100:
    WriteData               := TRUE;
END_CASE


fbFileOpen(
	sNetId:= , 
	sPathName:= sFileName, 
	nMode:= FOPEN_MODEAPPEND, 
	ePath:= PATH_GENERIC, 
	bExecute:= , 
	tTimeout:= T#10S, 
	bBusy=> , 
	bError=> , 
	nErrId=> , 
	hFile=> );

fbFileWrite(
	sNetId:= , 
	hFile:= fbFileOpen.hFile, 
	pWriteBuff:= ADR(sWriteData), 
	cbWriteLen:= StringLen(ADR(sWriteData)), 
	bExecute:= , 
	tTimeout:= T#10S, 
	bBusy=> , 
	bError=> , 
	nErrId=> nErrorWrite, 
	cbWrite=> );

fbFileClose(
	sNetId:= , 
	hFile:= fbFileOpen.hFile, 
	bExecute:= , 
	tTimeout:= T#10S, 
	bBusy=> , 
	bError=> , 
	nErrId=> );

bErrorWrite := fbFileOpen.bError OR fbFileWrite.bError;
END_METHOD

END_PROGRAM

// ---- APPLICATION/MAIN_APP.TcPOU
PROGRAM MAIN_APP
VAR
  eInit             : E_PROGRESS;   // application startup state info

  nProcess          : UINT;

  bNext             : BOOL := TRUE;
  bEnter            : BOOL := TRUE;
  bLeave            : BOOL := TRUE;

  tProcess          : array[1..MAX_PROCESS] of time;
END_VAR

//-----------------------------------------------------------------------------------------------------------------
//-----------------------------------------------------------------------------------------------------------------
// check for MAIN.eInit
//  - wait for fb_TransportUnit to be fully started up
//-----------------------------------------------------------------------------------------------------------------
IF NOT (MAIN.eInit = E_PROGRESS.PROGRESS_DONE) THEN eInit   := E_PROGRESS.PROGRESS_INVALID; RETURN; END_IF
//-----------------------------------------------------------------------------------------------------------------
//-----------------------------------------------------------------------------------------------------------------
//-----------------------------------------------------------------------------------------------------------------
// /assign dataflow
//-----------------------------------------------------------------------------------------------------------------
FOR nProcess := 1 TO MAX_PROCESS
DO
  GVL_APPLICATION.Simulation[nProcess].StationCtrl   := ADR(GVL_XTS.StationCtrl);
  GVL_APPLICATION.Simulation[nProcess].StationState  := ADR(GVL_XTS.StationState);

  GVL_APPLICATION.Simulation[nProcess].ProcessTime   := tProcess[nProcess];
END_FOR
//-----------------------------------------------------------------------------------------------------------------
//-----------------------------------------------------------------------------------------------------------------
Init();
//-----------------------------------------------------------------------------------------------------------------
//-----------------------------------------------------------------------------------------------------------------
// react to operation modes
//-----------------------------------------------------------------------------------------------------------------
//-----------------------------------------------------------------------------------------------------------------
CASE GVL_XTS.XtsTransportCtrl.Cmd
OF
  E_XTS_TRANSPORT_CTRL.CMD_INIT:

    FOR nProcess := 1 TO MAX_PROCESS
    DO
      GVL_APPLICATION.Simulation[nProcess].Init(); // clearing of XtsStations and Simulation
    END_FOR
END_CASE

CASE (GVL_XTS.XtsTransportState.State MOD E_PROGRESS.PROGRESS_DONE)
OF
  E_XTS_TRANSPORT_STATE.TRANSPORT_INIT:
    FOR nProcess := 1 TO MAX_PROCESS
    DO
      GVL_APPLICATION.Simulation[nProcess].Disable(); // switch off XtsStations and clear Simulation

      GVL_APPLICATION.Simulation[nProcess].EnableProcess := 0;
      GVL_APPLICATION.Simulation[nProcess].MoverEnter    := FALSE;
      GVL_APPLICATION.Simulation[nProcess].MoverOut      := FALSE;

      GVL_APPLICATION.Simulation[nProcess].Cycle();
    END_FOR

  E_XTS_TRANSPORT_STATE.TRANSPORT_START:
    FOR nProcess := 1 TO MAX_PROCESS
    DO
      GVL_APPLICATION.Simulation[nProcess].Next(bNext);

      IF (GVL_APPLICATION.Simulation[nProcess].StationCount > 0)
      THEN
        GVL_APPLICATION.Simulation[nProcess].EnableProcess := TO_WORD(EXPT(2,GVL_APPLICATION.Simulation[nProcess].StationCount))-1;
        GVL_APPLICATION.Simulation[nProcess].MoverEnter    := bEnter;
        GVL_APPLICATION.Simulation[nProcess].MoverOut      := bLeave;

      END_IF
      GVL_APPLICATION.Simulation[nProcess].Cycle();
    END_FOR
END_CASE

ACTION Init:
CASE eInit
OF
  E_PROGRESS.PROGRESS_INVALID:          // startup procedure for your application
    eInit                               := E_PROGRESS.PROGRESS_INIT;


  E_PROGRESS.PROGRESS_INIT:
      nProcess                                        := 1;
      tProcess[nProcess]                              := T#200MS;

      GVL_APPLICATION.Simulation[nProcess].StationFirst  := 1; // STN_12
      GVL_APPLICATION.Simulation[nProcess].StationLast   := 1;

      GVL_APPLICATION.Simulation[nProcess].TargetFirst   := 2;
      GVL_APPLICATION.Simulation[nProcess].TargetLast    := 5;
      GVL_APPLICATION.Simulation[nProcess].TargetMask    := 2#0001; // mask for target station

      //---------------------------------------------------------
      nProcess                                        := 2;
      tProcess[nProcess]                              := T#900MS;

      GVL_APPLICATION.Simulation[nProcess].StationFirst  := 2; // STN_01(1)
      GVL_APPLICATION.Simulation[nProcess].StationLast   := 5; // STN_01(4)

      GVL_APPLICATION.Simulation[nProcess].TargetFirst   := 6;
      GVL_APPLICATION.Simulation[nProcess].TargetLast    := 7;
      GVL_APPLICATION.Simulation[nProcess].TargetMask    := 2#0011; // mask for target station

      //---------------------------------------------------------
      nProcess                                        := 3;
      tProcess[nProcess]                              := T#335MS;

      GVL_APPLICATION.Simulation[nProcess].StationFirst  := 6; // STN_02(1)
      GVL_APPLICATION.Simulation[nProcess].StationLast   := 7; // STN_02(2)

      GVL_APPLICATION.Simulation[nProcess].TargetFirst   := 8;
      GVL_APPLICATION.Simulation[nProcess].TargetLast    := 8;
      GVL_APPLICATION.Simulation[nProcess].TargetMask    := 2#0001; // mask for target station

      //---------------------------------------------------------
      nProcess                                        := 4;
      tProcess[nProcess]                              := T#0MS;

      GVL_APPLICATION.Simulation[nProcess].StationFirst  := 8; // STN_03
      GVL_APPLICATION.Simulation[nProcess].StationLast   := 8;

      GVL_APPLICATION.Simulation[nProcess].TargetFirst   := 9;
      GVL_APPLICATION.Simulation[nProcess].TargetLast    := 10;
      GVL_APPLICATION.Simulation[nProcess].TargetMask    := 2#0011; // mask for target station

      //---------------------------------------------------------
      nProcess                                        := 5;
      tProcess[nProcess]                              := T#300MS;

      GVL_APPLICATION.Simulation[nProcess].StationFirst  := 9; // STN_04
      GVL_APPLICATION.Simulation[nProcess].StationLast   := 10;// STN_05

      GVL_APPLICATION.Simulation[nProcess].TargetFirst   := 11;
      GVL_APPLICATION.Simulation[nProcess].TargetLast    := 14;
      GVL_APPLICATION.Simulation[nProcess].TargetMask    := 2#0001; // mask for target station

      //---------------------------------------------------------
      nProcess                                        := 6;
      tProcess[nProcess]                              := T#2000MS;

      GVL_APPLICATION.Simulation[nProcess].StationFirst  := 11; // STN_06(1)
      GVL_APPLICATION.Simulation[nProcess].StationLast   := 14; // STN_06(4)

      GVL_APPLICATION.Simulation[nProcess].TargetFirst   := 15;
      GVL_APPLICATION.Simulation[nProcess].TargetLast    := 15;
      GVL_APPLICATION.Simulation[nProcess].TargetMask    := 2#0011; // mask for target station

      //---------------------------------------------------------
      nProcess                                        := 7;
      tProcess[nProcess]                              := T#150MS;

      GVL_APPLICATION.Simulation[nProcess].StationFirst  := 15; // STN_07
      GVL_APPLICATION.Simulation[nProcess].StationLast   := 15;

      GVL_APPLICATION.Simulation[nProcess].TargetFirst   := 16;
      GVL_APPLICATION.Simulation[nProcess].TargetLast    := 16;
      GVL_APPLICATION.Simulation[nProcess].TargetMask    := 2#0001; // mask for target station

      //---------------------------------------------------------
      nProcess                                        := 8;
      tProcess[nProcess]                              := T#350MS;

      GVL_APPLICATION.Simulation[nProcess].StationFirst  := 16; // STN_08
      GVL_APPLICATION.Simulation[nProcess].StationLast   := 16;

      GVL_APPLICATION.Simulation[nProcess].TargetFirst   := 17;
      GVL_APPLICATION.Simulation[nProcess].TargetLast    := 17;
      GVL_APPLICATION.Simulation[nProcess].TargetMask    := 2#0001; // mask for target station

      //---------------------------------------------------------
      nProcess                                        := 9;
      tProcess[nProcess]                              := T#300MS;

      GVL_APPLICATION.Simulation[nProcess].StationFirst  := 17; // STN_09
      GVL_APPLICATION.Simulation[nProcess].StationLast   := 17;

      GVL_APPLICATION.Simulation[nProcess].TargetFirst   := 18;
      GVL_APPLICATION.Simulation[nProcess].TargetLast    := 18;
      GVL_APPLICATION.Simulation[nProcess].TargetMask    := 2#0001; // mask for target station

      //---------------------------------------------------------
      nProcess                                        := 10;
      tProcess[nProcess]                              := T#0MS;

      GVL_APPLICATION.Simulation[nProcess].StationFirst  := 18; // STN_10
      GVL_APPLICATION.Simulation[nProcess].StationLast   := 18;

      GVL_APPLICATION.Simulation[nProcess].TargetFirst   := 19; // STN_11(1)
      GVL_APPLICATION.Simulation[nProcess].TargetLast    := 22; // STN_11(4)
      GVL_APPLICATION.Simulation[nProcess].TargetMask    := 2#0001; // mask for target station

      //---------------------------------------------------------
      nProcess                                        := 11;
      tProcess[nProcess]                              := T#1125MS;

      GVL_APPLICATION.Simulation[nProcess].StationFirst  := 19; // STN_11(1)
      GVL_APPLICATION.Simulation[nProcess].StationLast   := 22;

      GVL_APPLICATION.Simulation[nProcess].TargetFirst   := 1; // STN_12
      GVL_APPLICATION.Simulation[nProcess].TargetLast    := 1;
      GVL_APPLICATION.Simulation[nProcess].TargetMask    := 2#0001; // mask for target station


    eInit                               := E_PROGRESS.PROGRESS_DONE;

END_CASE
END_ACTION

END_PROGRAM

// ---- APPLICATION/fb_Simulation.TcPOU
//---------------------------------------------------------------------------------------------------------------
//
//  HAUD 2023.03.27
//
//
//  fb_Simulation
//
//    !!! NOT FOR USE IN PRODUCTION !!! --> build something from your mind, this gets messy if you do not
//
//  - grouping of xts stations to sync start process
//  - nFirst to nLast xts stations are checked for starting process simultaneously
//  - basic preparation of station target index in PrepareTarget()
//  - handshake with station control for mover transport through station
//
//---------------------------------------------------------------------------------------------------------------
// This SOFTWARE is provided as an Exemple by THE PROVIDER "as is" and "with all faults." THE PROVIDER makes no 
// representations or warranties of any kind concerning the safety, suitability, lack of viruses, inaccuracies, 
// typographical errors, or other harmful components of this SOFTWARE. There are inherent dangers in the use of 
// any software, and you are solely responsible for determining whether this SOFTWARE is compatible with your 
// equipment and other software installed on your equipment. You are also solely responsible for the protection 
// of your equipment and backup of your data, and THE PROVIDER will not be liable for any damages you may suffer 
// in connection with using, modifying, or distributing this SOFTWARE.
//---------------------------------------------------------------------------------------------------------------
FUNCTION_BLOCK fb_Simulation
VAR
  _sCheck                     : STRING;
  _tonProcess                 : Tc2_Standard.TON;
  _tProcess                   : TIME := T#500MS;

  _AllStationMoverPerMinute   : UINT;
  _tonPartsPerMinute          : Tc2_Standard.TON;

  {attribute 'displaymode':='bin'}
  _wEnter                     : WORD;
  {attribute 'displaymode':='bin'}
  _wStart                     : WORD;
  {attribute 'displaymode':='bin'}
  _wOut                       : WORD;
  {attribute 'displaymode':='bin'}
  _wGone                      : WORD;
  {attribute 'displaymode':='bin'}
  _wEnableProcess             : WORD; // bits switch on stations

  {attribute 'displaymode':='bin'}
  _TargetMask                 : BYTE;

  _stCtrl                     : POINTER TO ARRAY[1..MAX_STATION]  OF ST_STATION_CTRL;
  _stState                    : POINTER TO ARRAY[1..MAX_STATION]  OF ST_STATION_STATE;

  // controlling bits from properties used on the outside
  _bNext,
  _bMoverEnter,
  _bMoverOut                  : BOOL;

  // who is included in process
  // _nFirst to _nLast MUST be in closed consecutive order
  _nProcessState,
  _nStation,
  _nStationCount,
  _nFirstStation,
  _nLastStation               : UINT;

  _nTarget,
  _nFirstTarget,
  _nLastTarget                : UINT;

  _nPreparedTarget            : ARRAY[1..MAX_MOVER]  OF UINT;

  _nMoverPerMinute,
  _nMoverCount,
  _nMoverCountOld             : ARRAY[1..MAX_STATION]  OF UINT;
END_VAR

METHOD Check : BOOL

IF (_nFirstStation < 1) OR
   (_nFirstStation > MAX_STATION)
THEN
  _sCheck                     := '_nFirstStation out of bounds';
  RETURN;
END_IF

IF (_nLastStation < 1) OR
   (_nLastStation > MAX_STATION)
THEN
  _sCheck                     := '_nLastStation out of bounds';
  RETURN;
END_IF

IF (_nFirstTarget < 1) OR
   (_nFirstTarget > MAX_STATION)
THEN
  _sCheck                     := '_nFirstTarget out of bounds';
  RETURN;
END_IF

IF (_nLastTarget < 1) OR
   (_nLastTarget > MAX_STATION)
THEN
  _sCheck                     := '_nLastTarget out of bounds';
  RETURN;
END_IF

IF NOT (_stCtrl  <> 0)
THEN
  _sCheck                     := '_stCtrl: missing pointer';
  RETURN;
END_IF

IF NOT (_stState <> 0)
THEN
  _sCheck                     := '_stState: missing pointer';
  RETURN;
END_IF


_sCheck                       := TO_STRING(E_PROGRESS.PROGRESS_DONE);
Check                         := TRUE;
END_METHOD

METHOD Cycle
VAR_INST
  _k                  : UINT;
  _rtrigProcess       : ARRAY[1..MAX_STATION] OF Tc2_Standard.R_TRIG;
END_VAR
IF NOT Check() THEN RETURN; END_IF

_nStationCount                              := _nLastStation - _nFirstStation + 1;

IF (_nStationCount < 1)
THEN
  RETURN;
END_IF

FOR _nStation := _nLastStation TO _nFirstStation BY(-1) 
DO
  CASE _stState^[_nStation].eState
  OF
    E_STATION_STATE.STATION_DISABLE,
    E_STATION_STATE.STATION_ENABLE, 
    E_STATION_STATE.STATION_DETECT_MOVER:
      _wOut    := _wGone                    := 0;
      _wEnter                               := DelBitWord(_wEnter, (_nStation-_nFirstStation));
      _wStart                               := DelBitWord(_wStart, (_nStation-_nFirstStation));
      IF (GetBitWord(_wEnableProcess, (_nStation-_nFirstStation)))
      THEN
        IF (_bMoverEnter)
        THEN
          _stCtrl^[_nStation].eCmd          := E_STATION_CTRL.STATION_ENABLE;
        ELSE
          _stCtrl^[_nStation].eCmd          := E_STATION_CTRL.STATION_DISABLE;
        END_IF
      ELSE
        _stCtrl^[_nStation].eCmd            := E_STATION_CTRL.STATION_DISABLE;
      END_IF


    E_STATION_STATE.STATION_MOVER_ENTER:
      _wEnter                               := SetBitWord(_wEnter, (_nStation-_nFirstStation));
      IF _bMoverEnter
      THEN
        _tonProcess(IN                      := FALSE, 
                    PT                      := _tProcess);

        _stCtrl^[_nStation].nTargetStation  := 0;
        _stCtrl^[_nStation].eCmd            := E_STATION_CTRL.STATION_MOVER_ENTER;
      END_IF

    E_STATION_STATE.STATION_PROCESS_START:
      _wEnter                               := DelBitWord(_wEnter, (_nStation-_nFirstStation));
      _wStart                               := SetBitWord(_wStart, (_nStation-_nFirstStation));
  
      // check if ALL XtsStations have mover in place to work
      IF (_wStart = TO_WORD(EXPT(2,_nStationCount))-1)
      THEN
        _tonProcess(IN                      := TRUE, 
                    PT                      := _tProcess);

        IF _tonProcess.Q
        THEN
          PrepareTargets(FALSE);
          _stCtrl^[_nStation].eCmd          := E_STATION_CTRL.STATION_PROCESS_DONE;
        END_IF
      END_IF

    E_STATION_STATE.STATION_CHECK_NEST:
      _wEnter                               := SetBitWord(_wEnter, (_nStation-_nFirstStation));
      _wStart                               := DelBitWord(_wStart, (_nStation-_nFirstStation));
      _tonProcess(IN                        := FALSE, 
                  PT                        := _tProcess);

      IF (_bNext)
      THEN
        // check if ALL XtsStations have nest to work
        IF (_wEnter = TO_WORD(EXPT(2,_nStationCount))-1)
        THEN
          _stCtrl^[_nStation].eCmd          := E_STATION_CTRL.STATION_MOVER_ENTER;
        END_IF
      END_IF


    E_STATION_STATE.STATION_MOVER_OUT:
      _wOut                                 := SetBitWord(_wOut, (_nStation-_nFirstStation));
      _tonProcess(IN                        := FALSE, 
                  PT                        := _tProcess);

      IF _bMoverOut
      THEN
        // nest mask for this mover in target station, sender decides what to work in target
        _stCtrl^[_nStation].nMask           := _TargetMask;

        // check if ALL XtsStations have mover to send
        IF (_wOut = TO_WORD(EXPT(2,_nStationCount))-1)
        THEN
          _nProcessState                    := 10;
        END_IF
      END_IF
  END_CASE
END_FOR

CASE _nProcessState
OF
10:
  // ctrl has to decide where to send mover; this depends on YOUR decision
  IF PrepareTargets(TRUE)
  THEN
    PrepareTargets(FALSE);
    _nProcessState                          := 30;
  END_IF
END_CASE
CASE _nProcessState
OF
30:
  FOR _nStation := _nLastStation TO _nFirstStation BY(-1) 
  DO
    IF _bNext
    THEN
      // start outfeed of mover
      _stCtrl^[_nStation].eCmd              := E_STATION_CTRL.STATION_MOVER_OUT;
    END_IF

    CASE _stState^[_nStation].eState
    OF
      E_STATION_STATE.STATION_MOVER_GONE:
        // whO is gone?
        _wGone                              := SetBitWord(_wGone, (_nStation-_nFirstStation));
    END_CASE
  END_FOR
  // check if ALL XtsStations are empty
  IF (_wGone = TO_WORD(EXPT(2,_nStationCount))-1)
  THEN
    _nProcessState                          := 40;
  END_IF
END_CASE
CASE _nProcessState
OF
40:
  _nProcessState                            := 0;
  FOR _nStation := _nLastStation TO _nFirstStation BY(-1) 
  DO
    // let XtsStations jump back to disable
    _stCtrl^[_nStation].eCmd                := E_STATION_CTRL.STATION_MOVER_GONE;
  END_FOR
END_CASE


//-----------------------------------------------------------------------------
// Mover per Minute counter all XtsStations in range
//-----------------------------------------------------------------------------
_AllStationMoverPerMinute   := 0; 
//-----------------------------------------------------------------------------
// mover counter
//-----------------------------------------------------------------------------
FOR _k := _nLastStation TO _nFirstStation BY(-1) 
DO
  _rtrigProcess[_k](CLK:= (_stCtrl^[_k].eCmd = E_STATION_CTRL.STATION_MOVER_OUT));

  IF _rtrigProcess[_k].Q
  THEN
    _nMoverCount[_k]         := _nMoverCount[_k] + 1;
  END_IF
  
  IF _tonPartsperMinute.Q
  THEN
    // count every XtsStation in range
    _nMoverPerMinute[_k]    := _nMoverCount[_k] - _nMoverCountOld[_k];
    _nMoverCountOld [_k]    := _nMoverCount[_k];
  END_IF
  // sum up all XtsStations in range
  _AllStationMoverPerMinute := _AllStationMoverPerMinute + _nMoverPerMinute[_k]; 
END_FOR

IF _tonPartsperMinute.q
THEN
  _tonPartsperMinute(IN:=FALSE);
END_IF

_tonPartsperMinute(IN:= TRUE, PT:= T#60S);
END_METHOD

METHOD PUBLIC DelBitWord : WORD
VAR_INPUT
  inVal   : WORD;
  bitNo   : DINT;
END_VAR
VAR
  wConst : WORD := 1;
END_VAR
IF ( inVal AND SHL( wConst,bitNo MOD 16 ) ) > 0 THEN
  DelBitWord := inVal XOR (SHL( wConst,bitNo MOD 16 ));
ELSE
  DelBitWord := inVal;
END_IF
END_METHOD

METHOD Disable : BOOL
VAR_INPUT
END_VAR
IF NOT (_nLastStation   > 0) OR
   NOT (_nFirstStation  > 0) OR
   NOT (_nLastStation   < MAX_STATION+1) OR
   NOT (_nFirstStation  < MAX_STATION+1)
THEN
  Disable := FALSE;
ELSE
  FOR _nStation := _nLastStation TO _nFirstStation BY(-1) 
  DO
    _stCtrl^[_nStation].eCmd              := E_STATION_CTRL.STATION_DISABLE;
    _stCtrl^[_nStation].nMask             := 0;
  END_FOR

  memset(ADR(_nMoverCount),    0, SIZEOF(_nMoverCount));
  memset(ADR(_nMoverCountOld), 0, SIZEOF(_nMoverCountOld));
  _nProcessState :=  _nTarget             := 0;
  
  Disable := TRUE;
END_IF
END_METHOD

PROPERTY EnableProcess : word
GET
EnableProcess := _wEnableProcess;
END_GET
SET
_wEnableProcess := EnableProcess;
END_SET
END_PROPERTY

METHOD PUBLIC GetBitWord : BOOL
VAR_INPUT
  inVal   : WORD;
  bitNo   : DINT;
END_VAR
VAR
  wConst : WORD := 1;
END_VAR
IF ( inVal AND SHL( wConst,DINT_TO_SINT(bitNo) MOD 16 ) ) > 0
THEN
  GetBitWord := TRUE;
ELSE
  GetBitWord := FALSE;
END_IF
END_METHOD

METHOD Init : BOOL
VAR_INPUT
END_VAR
IF NOT (_nLastStation   > 0) OR
   NOT (_nFirstStation  > 0) OR
   NOT (_nLastStation   < MAX_STATION+1) OR
   NOT (_nFirstStation  < MAX_STATION+1)
THEN
  Init := FALSE;
ELSE
  FOR _nStation := _nLastStation TO _nFirstStation BY(-1) 
  DO
    _stCtrl^[_nStation].eCmd              := E_STATION_CTRL.STATION_INIT;
    _stCtrl^[_nStation].nMask             := 0;
  END_FOR

  memset(ADR(_nMoverCount),    0, SIZEOF(_nMoverCount));
  memset(ADR(_nMoverCountOld), 0, SIZEOF(_nMoverCountOld));
  _nProcessState :=  _nTarget             := 0;
  
